// TwinCAT 3 PLC project BMS_PTM
// ProgramVersion: 3.1.4023.0
// libraries:
//   EfficientIO Communicator, * (EfficientIO)
//   Lynus Energy Basic, * (Lynus AG)
//   Lynus Energy ModbusTCP, * (Lynus AG)
//   Lynus Persistent Data V1, * (Lynus AG)
//   Lynus Standards, * (Lynus AG)
//   Tc2_ModbusSrv, * (Beckhoff Automation GmbH)
//   Tc2_Standard, * (Beckhoff Automation GmbH)
//   Tc2_System, * (Beckhoff Automation GmbH)
//   Tc2_Utilities, * (Beckhoff Automation GmbH)
//   Tc3_IotBase, * (Beckhoff Automation GmbH)
//   Tc3_Module, * (Beckhoff Automation GmbH)
// project tree:
//   / FastTask.TcTTO (not stored), MiddleTask.TcTTO, SlowTask.TcTTO (not stored)
//   FB/ FB_BatteryInverter_T.TcPOU, FB_Convert_Huawei_SmartLogger.TcPOU (not stored) (excluded from build), FB_EMS_T.TcPOU, FB_EMS_T_1.TcPOU (excluded from build), FB_EM_Beckhoff_KL3403.TcPOU (not stored), FB_Huawei_SmartLogger_1.TcPOU (excluded from build), FB_IntervalBit.TcPOU (not stored), FB_MqttCommunicator_V2_1.TcPOU (not stored), FB_Xelectrix_Powerbox_T.TcPOU
//   POUs/ prgAD.TcPOU, prgBattery.TcPOU, prgComEffIO.TcPOU, prgGrid.TcPOU, prgEMS.TcPOU, prgHouse.TcPOU, prgPersistent.TcPOU, prgPV.TcPOU, prgRWEffIO.TcPOU, prgVarEffIO.TcPOU (not stored), prg_SystemTime.TcPOU (not stored)
// real-time tasks:
//   TASK FastTask: cycle T#5ms, priority 19, ADS port 350
//   TASK MiddleTask: cycle T#10ms, priority 20, ADS port 351
//   TASK SlowTask: cycle T#20ms, priority 21, ADS port 352
// I/O:
//   DEVICE Device 1 (Beckhoff CCAT)
//   DEVICE Device 2 (CX-BK)
//     Box 1 (CX-BK)
// variable links:
//   BMS_PTM/BMS_PTM Instance <-> Device 2 (CX-BK)/Box 1 (CX-BK)
//     MiddleTask Inputs/prgGrid.fbEM1.fbKL3403.byStateCH1 <-> Term 2 (KL3403)/Channel 1/State
//     MiddleTask Inputs/prgGrid.fbEM1.fbKL3403.byStateCH2 <-> Term 2 (KL3403)/Channel 2/State
//     MiddleTask Inputs/prgGrid.fbEM1.fbKL3403.byStateCH3 <-> Term 2 (KL3403)/Channel 3/State
//     MiddleTask Inputs/prgGrid.fbEM1.fbKL3403.iDataInCH1 <-> Term 2 (KL3403)/Channel 1/Data In
//     MiddleTask Inputs/prgGrid.fbEM1.fbKL3403.iDataInCH2 <-> Term 2 (KL3403)/Channel 2/Data In
//     MiddleTask Inputs/prgGrid.fbEM1.fbKL3403.iDataInCH3 <-> Term 2 (KL3403)/Channel 3/Data In
//     MiddleTask Inputs/prgGrid.fbKBusState.uiKBusState_OUT <-> Inputs/State
//     MiddleTask Outputs/prgGrid.fbEM1.fbKL3403.byCntrCH1 <-> Term 2 (KL3403)/Channel 1/Ctrl
//     MiddleTask Outputs/prgGrid.fbEM1.fbKL3403.byCntrCH2 <-> Term 2 (KL3403)/Channel 2/Ctrl
//     MiddleTask Outputs/prgGrid.fbEM1.fbKL3403.byCntrCH3 <-> Term 2 (KL3403)/Channel 3/Ctrl

CONFIGURATION BMS_PTM
    RESOURCE PLC ON TwinCAT3
        TASK MiddleTask(INTERVAL := T#10ms, PRIORITY := 20);
        PROGRAM prgBattery WITH MiddleTask : prgBattery;
        PROGRAM prgGrid WITH MiddleTask : prgGrid;
        PROGRAM prgHouse WITH MiddleTask : prgHouse;
        PROGRAM prgPersistent WITH MiddleTask : prgPersistent;
        PROGRAM prgEMS WITH MiddleTask : prgEMS;
        PROGRAM prgPV WITH MiddleTask : prgPV;
        PROGRAM prgAD WITH MiddleTask : prgAD;
    END_RESOURCE
END_CONFIGURATION

// ---- POUs/prgBattery.TcPOU
PROGRAM prgBattery
VAR PERSISTENT
	bEnableBattery				: BOOL;							//{#lynus.ag#()}
	byPrioBattery				: BYTE;							//{#lynus.ag#()}
	lrMaxCapacityBattery		: LREAL;						//{#lynus.ag#()}
	lrCounterBattProd			: LREAL;						//{#lynus.ag#()}
	lrCounterBattCons			: LREAL;						//{#lynus.ag#()}
END_VAR
VAR
	fbBattery					: FB_Xelectrix_Powerbox_T;
	fbBattCounter				: FB_EnergyCounter;
	bIsEnabledBattery			: BOOL;							//{#lynus.ag#()}
	bResetBattery				: BOOL;							//{#lynus.ag#()}
	bSResetBattery				: BOOL;							//{#lynus.ag#()}
	byErrorWarningBattery		: BYTE;							//{#lynus.ag#()}
	dwSOCBattery				: DWORD;						//{#lynus.ag#()}
	rTargetPowerBattery			: REAL;							//{#lynus.ag#()}
	lrPowerBattery				: LREAL;						//{#lynus.ag#()}
	lrActualCapacityBattery		: LREAL;						//{#lynus.ag#()}
	lrEnergyConsumption			: LREAL;						//{#lynus.ag#()}
	lrEnergyProduction			: LREAL;						//{#lynus.ag#()}
	mTest: BOOL;

	lrPowerBattery2				: LREAL;
	lrPowerBattery3				: LREAL;						

	int_GridState: INT;											//{#lynus.ag#()}
	int_BatteryState: INT;										//{#lynus.ag#()}
	int_OperatingState: INT;									//{#lynus.ag#()}
	int_ErrorState: INT;										//{#lynus.ag#()}

	FB_Interval: FB_IntervalBit;
	m_IslandOperationStart: BOOL;								//{#lynus.ag#()}
	m_IslandOperationOngoing: BOOL;								//{#lynus.ag#()}
	m_IslandOperationStop: BOOL;								//{#lynus.ag#()}
	t_Interval :TIME:=T#30M;
	t_HightTime :TIME:=T#1S;
	
	
	m_BatteryErrorActive: BOOL;									//{#lynus.ag#()}
	m_BatteryModbusCommError: BOOL;								//{#lynus.ag#()}
	m_BatteryTargetSPError: BOOL;								//{#lynus.ag#()}
	Ton_Delay_BatteryError: Ton;
	Ton_Delay_BatteryModbusError: Ton;
	Ton_Delay_BatterySPError: Ton;
END_VAR

IF mtest THEN
	Lynus_Standards.GVL_Energy.stDataOfBatteryInverters[1,1].rTargetPowerEMS:=0;
	mtest:=FALSE;
 END_IF
 
fbBattery(
	bEnable:= bEnableBattery, 
	bActivateControl:= TRUE, 
	byUnitID:= 1, 
	byPriority:= byPrioBattery, 
	diNrOfEMS_IN:= prgEMS.fbEMS.diNrOfEMS_OUT, 
	lrMaxCapacityBattery:= lrMaxCapacityBattery, 
	sIPAdress:= '192.168.66.240', 						// modify IP Adress
	bReset:= bResetBattery, 
	stDataXelectrix=> , 
	stDataBatt=> , 
	stDataBattInverter=> , 
	stDataEMPower_Grid=> , 
	stDataEMCounter_Grid=> , 
	diNrOfBatt_OUT=> , 
	diNrOfBattInverter_OUT=> , 
	diNrOfEM_OUT_Grid=> , 
	lrMaxCapacityBattery_OUT=> );
	
//Out
bIsEnabledBattery 		:= fbBattery.stDataBatt.bEnabled;
bSResetBattery			:= fbBattery.stDataBattInverter.bStateReset;
dwSOCBattery 			:= fbBattery.stDataBatt.dwSOC;
rTargetPowerBattery 	:= fbBattery.stDataBattInverter.rTargetPower;
lrPowerBattery 			:= fbBattery.stDataBatt.lrPower;
lrActualCapacityBattery := fbBattery.lrMaxCapacityBattery_OUT;	
byErrorWarningBattery 	:= fbBattery.stDataBatt.byErrorWarning;
lrEnergyConsumption		:= fbBattery.fbEMGrid.lrTotalCounterEnergy_Consumption;
lrEnergyProduction		:= fbBattery.fbEMGrid.lrTotalCounterEnergy_Production;					
lrPowerBattery2			:= fbBattery.fbEMGrid.lrPowerTotal/1000;
							
// EnergyCounter
fbBattCounter(
	byActiveTariff:= 1, 
	lrPowerInput:= lrPowerBattery, 
	lrTotalCounterEnergy_Consumption=> , 
	lrTotalCounterEnergy_Production=> , 
	lrCounterEnergyT1_Consumption=> , 
	lrCounterEnergyT2_Consumption=> , 
	lrCounterEnergyT1_Production=> , 
	lrCounterEnergyT2_Production=> );
	
IF fbBattCounter.lrTotalCounterEnergy_Production > lrCounterBattProd THEN  	
	lrCounterBattProd := fbBattCounter.lrTotalCounterEnergy_Production;
END_IF

IF fbBattCounter.lrTotalCounterEnergy_Consumption > lrCounterBattCons THEN  	
	lrCounterBattCons := fbBattCounter.lrTotalCounterEnergy_Consumption;
END_IF

// send e states to cloud
int_GridState 		:= fbBattery.stDataXelectrix.eGridState;
int_BatteryState	:= fbBattery.stDataXelectrix.eBatteryState;
int_OperatingState	:= fbBattery.stDataXelectrix.eOperatingState;
int_ErrorState		:= fbBattery.stDataXelectrix.eErrorState;


// create bits when battery is in island operation

FB_Interval(
	m_Input			:=  prgBattery.fbBattery.stDataXelectrix.eGridState = 2,	//   2 = Island Mode 
	t_Interval 		:= t_Interval , 
	t_HighTime		:= t_HightTime, 
	m_RisingEdge	=> m_IslandOperationStart, 
	m_Interval		=> m_IslandOperationOngoing, 
	m_FallingEdge	=> m_IslandOperationStop);

// monitoring Battery status

Ton_Delay_BatteryError (In := fbBattery.stDataXelectrix.eErrorState =2,
						PT :=T#5S,
						Q => m_BatteryErrorActive);

Ton_Delay_BatteryModbusError (	In := fbBattery.stDataXelectrix.eErrorState = 1,
								PT :=T#10M,
								Q => m_BatteryModbusCommError);						

Ton_Delay_BatterySPError (	In := ABS(fbBattery.iSetpointPower/10-lrPowerBattery) > 20 AND fbBattery.stDataXelectrix.eGridState<>2 AND fbBattery.stDataBatt.dwSOC<90,	// not alarming during island operation
							PT :=T#1M,
							Q => m_BatteryTargetSPError);

END_PROGRAM

// ---- FB/FB_Xelectrix_Powerbox_T.TcPOU
FUNCTION_BLOCK FB_Xelectrix_Powerbox_T
VAR_INPUT PERSISTENT
	bEnable							: BOOL;											//{#lynus.ag#()} //True = Function is enabled, FALSE = Function is dissabled, no new Data
	bActivateControl				: BOOL;											//Activate the control from the Xelectrix Inverter over Modbus TCP (False = Inverter work by himself)
	byUnitID						: BYTE;											//Unit ID fromt the Inverter (0 to 255)
	byPriority						: BYTE;											//{#lynus.ag#()} //Priority of the Device
	diNrOfEMS_IN					: DINT;											//Number of EMS what control this Device.
	lrMaxCapacityBattery			: LREAL;										//{#lynus.ag#()} //Max Capacity from the Battery in kWh. Here on this Function this Input Value cames from Inside of the Function.
	sIPAdress						: STRING(15);									//IP Adress from the Inverter
END_VAR
VAR_INPUT
	bReset							: BOOL;											//{#lynus.ag#()} //Reset the device after a Error or a Warning
END_VAR
VAR_OUTPUT
	stDataXelectrix					: ST_Xelectrix_Powerbox_OutData;				//Shows the specific output data from the Xelectric device
	stDataBatt						: ST_Battery_Output;							//{#lynus.ag#()} //Output structure with Data from Battery
	stDataBattInverter				: ST_BatteryInverter_Output;					//{#lynus.ag#()} //Output structure with Data from Battery Inverter
	stDataEMPower_Grid				: ST_ElectricMeter_Output_Power;				//Output structure with Data from Electric Meter Grid (Power Data)
	stDataEMCounter_Grid			: ST_ElectricMeter_Output_Counter;				//Output structure with Data from Electric Meter Grid (Counter Data)
	diNrOfBatt_OUT					: DINT;											//Active Number from the Battery Function for using on other functions
	diNrOfBattInverter_OUT			: DINT;											//Active Number from the Battery Inverter Function for using on other functions
	diNrOfEM_OUT_Grid				: DINT;											//Active Number from the Electric Meter for using on other functions
	lrMaxCapacityBattery_OUT		: LREAL;										//Max kWh from the Battery system. The Xelectrix System deliver this value.
END_VAR
VAR

	fbBattery						: FB_Battery;									//Function block for battery

	fbBatteryInverter				: FB_BatteryInverter_T;							//Function block for battery inveter

	fbEMGrid						: FB_ElectricMeter;								//Electric Meter Function 

	fbPIDChrgStandby				: FB_PID;										//Controller to control the battery current on 0 in the standby mode	

	fbNumberDeviceBattery			: FB_NumberOfDevice;							//Function block to calcualte the number of the Device

	fbNumberDeviceBatteryInvert		: FB_NumberOfDevice;							//Function block to calcualte the number of the Device

	fbNumberDeviceGrid				: FB_NumberOfDevice;							//Function block to calcualte the number of the Device

	fbMBRead_FC3					: FB_MBReadRegs;								//Modbus Read Function (FC3)

	fbMBWrite_FC16					: FB_MBWriteRegs;								//Modbus Write Function (FC16)

	fbConvertData					: FB_CV_WORD_TO_DWORD;							//Convert 2 Words in a Dword

	timDelay						: TON;											//Timer for Delay between Requests

	timTimeout						: TON;											//Timer for Timeout

	timDissableFunctions			: TON;											//Timer to dissable the Function after Lynus_Standards.Constants_General.tTimeDissableLynusFunctions Days without connection to the Lynus Cloud

	timResetConnectionOnGVL			: TON;											//Timer to try reset the connection Flag on the GVL. (When somebody delete the Connection Function and make only a onlinechange)

	timReset						: TON;											//Timer to reset the Inverter after a Error

	timErrorMTCP					: TON;											//Delay when Error on Modbus TCP

	timSetStandbyCntrl				: TOF;											//Timer to set the Standby Controller

	FPEnable						: R_TRIG;										//Internal positive Edge

	FPError_FC_3					: R_TRIG;										//Internal positive Edge

	FPError_FC_16					: R_TRIG;										//Internal positive Edge

	FPActivateControl				: R_TRIG;										//Internal positive Edge

	FNTimDissable					: F_TRIG;										//Internal negative Edge

	PD_String						: FB_PersistentData_String;						//Function to save persistent data

	arrPD							: ARRAY[1..7] OF FB_PersistentData_Number;		//Function to save persistent data

	arrBuffer_FC3					: ARRAY[1..48] OF WORD;							//Buffer with Data from FC3

	arrBuffer_FC16					: ARRAY[1..2] OF WORD;							//Buffer with Data from FC16

	arrCounterForGVL				: ARRAY[1..3] OF DINT;							//Counter to clean old data on GVL

	bEnergyGridConsReceived			: BOOL;											//Energy Consumption from Grid first time received

	bEnergyGridProdReceived			: BOOL;											//Energy Production from Grid first time received

	byWaitInStep					: BYTE;											//Wait in Step before start to clean data on PLC

	byLPWorkAroundACDevice			: BYTE;											//Loop for Workaround

	byNumberOfZero					: BYTE;											//Number with 0 Value from AC Messurement

	iSetpointPower					: INT;											//Power Setpoint in W

	iStateGVLData					: INT;											//State machine to handle the data on the GVL

	iStateModbusRead				: INT;											//State variable for Statemachine

	iStateModbusWrite				: INT;											//State variable for Statemachine

	iStateModbusError				: INT;											//State variable for Statemachine

	iStateModbus_CP					: INT;											//Compare State variable

	iMaxDcDischargeCurrentBattery	: INT;											//Variable to convert from negative to positive value

	diLPForGVL						: DINT;											//Loop to clean old data on GVL

	lrEnergyGridConsumption_CP		: LREAL;										//Energy Consumption from Grid for calculation for Workaround why Xelectrix send sometimes big value 

	lrEnergyGridProduction_CP		: LREAL;										//Energy Production from Grid for calculation for Workaround why Xelectrix send sometimes big value 
	realTemp: REAL;
END_VAR
VAR PERSISTENT
	{attribute 'conditionalshow'}
	diNrOfEMS_IN_CP					: DINT;											//Number of EMS what control this Device to compare with the original
END_VAR

//Creator : Kai Ebensperger
//Company : Lynus AG
//Date : 30.06.2021
//Version : 1.0.0.0

//With this function its possible to read out values from the Xelectrix Powerbox from the factory Xelectrix
//Its also possible to controll the power in and out from Battery if its necessary.
//The protocol to the Inverter/powerbox is Modbus TCP
//When this Function is not enabled, then the Inverter is not off. But no power flows into or out of the battery.
//This Inverter deliver also the Grid power (smart Meter).
//Versions that are supported : 106
//NOTE : This Function block not support the complete emergency power mode. He switch not off when the byMaxDepthOfDischargeEPO is reached because this make the inverter by himself.

//NOTE for diNr.....Designation => 
//_IN = Here Data come in from other Functions or go out to other functions about the GVL
//_OUT = Here Data go out to other functions about the GVL

(*------------------------------------------------------------------------------------------General Input Part---------------------------------------------------------------------------------------------*)

//Check limitation
diNrOfEMS_IN := LIMIT(0,diNrOfEMS_IN,Constants_Energy.diMaxNumberOfEMS);
	
(*-------------------------------------------------------------Calcualte the number of Battery system---------------------------------------------------------------*)

fbNumberDeviceBattery(
	diActualNumberOfDevices:= Lynus_Standards.GVL_Energy.stNumberOfDevices.diNumberOfBatterys, 
	diMaxNumberOfDevices:= Constants_Energy.diMaxNumberOfBatterys, 
	udiCounterOnlineChange:= TwinCAT_SystemInfoVarList._AppInfo.OnlineChangeCnt, 
	bNumberIsCalculatet=> , 
	bFPNumberIsCalculatet=> , 
	bOnlineChange=> , 
	diNumberForThisDevice=> diNrOfBatt_OUT, 
	diNumberOfTotalDevices=> );

//Write new Numer on GVL
IF fbNumberDeviceBattery.bFPNumberIsCalculatet THEN
	Lynus_Standards.GVL_Energy.stNumberOfDevices.diNumberOfBatterys := fbNumberDeviceBattery.diNumberOfTotalDevices;	
END_IF

//Delete old Number on GVL
IF fbNumberDeviceBattery.bOnlineChange THEN 
	Lynus_Standards.GVL_Energy.stNumberOfDevices.diNumberOfBatterys := diNrOfBatt_OUT;	
		iStateGVLData := 1; 
END_IF

fbNumberDeviceBatteryInvert(
	diActualNumberOfDevices:= Lynus_Standards.GVL_Energy.stNumberOfDevices.diNumberOfBatteryInverters, 
	diMaxNumberOfDevices:= Constants_Energy.diMaxNumberOfBatteryInverters, 
	udiCounterOnlineChange:= TwinCAT_SystemInfoVarList._AppInfo.OnlineChangeCnt, 
	bNumberIsCalculatet=> , 
	bFPNumberIsCalculatet=> , 
	bOnlineChange=> , 
	diNumberForThisDevice=> diNrOfBattInverter_OUT, 
	diNumberOfTotalDevices=> );

//Write new Numer on GVL
IF fbNumberDeviceBatteryInvert.bFPNumberIsCalculatet THEN
	Lynus_Standards.GVL_Energy.stNumberOfDevices.diNumberOfBatteryInverters := fbNumberDeviceBatteryInvert.diNumberOfTotalDevices;	
END_IF

//Delete old Number on GVL
IF fbNumberDeviceBatteryInvert.bOnlineChange THEN 
	Lynus_Standards.GVL_Energy.stNumberOfDevices.diNumberOfBatteryInverters := diNrOfBattInverter_OUT;	
		iStateGVLData := 1; 
END_IF

fbNumberDeviceGrid(
	diActualNumberOfDevices:= Lynus_Standards.GVL_Energy.stNumberOfDevices.diNumberOfElectricMeters, 
	diMaxNumberOfDevices:= Constants_Energy.diMaxNumberOfElectricMeters, 
	udiCounterOnlineChange:= TwinCAT_SystemInfoVarList._AppInfo.OnlineChangeCnt, 
	bNumberIsCalculatet=> , 
	bFPNumberIsCalculatet=> , 
	bOnlineChange=> , 
	diNumberForThisDevice=> diNrOfEM_OUT_Grid, 
	diNumberOfTotalDevices=> );

//Write new Numer on GVL
IF fbNumberDeviceGrid.bFPNumberIsCalculatet THEN
	Lynus_Standards.GVL_Energy.stNumberOfDevices.diNumberOfElectricMeters := fbNumberDeviceGrid.diNumberOfTotalDevices;	
END_IF			

(*-------------------------------------------------------------Service from Backend is ready and check the connection to backend for dissabel/enable Function---------------------------------------------------------------*)

//Try to reset the variable for connection on the GVL. When all is normal then the Lynus Mqtt connection function set this variable to true in the next cycle
//When we have no connection to the backend then after Lynus_Standards.Constants_General.tTimeDissableLynusFunctions days the Function is dissabled with all of his functionalities
timResetConnectionOnGVL(IN:= NOT timResetConnectionOnGVL.Q, PT:= T#1H, Q=> , ET=> );
	IF timResetConnectionOnGVL.Q THEN Lynus_Standards.GVL_Communicator.bStateConnectionToEnableFunctions := FALSE; END_IF
		IF NOT Lynus_Standards.GVL_Communicator.bStateConnectionToEnableFunctions THEN timDissableFunctions.IN := TRUE; ELSE timDissableFunctions.IN := FALSE; END_IF  
			timDissableFunctions(IN:= , PT:= Lynus_Standards.Constants_General.tTimeDissableLynusFunctions, Q=> , ET=> );
			
(*------------------------------------------------------------------------------------------State Machine Read---------------------------------------------------------------------------------------------*)

//When the function is not enabled then the fronius control by himself without modbus tcp connection
IF NOT bEnable OR timDissableFunctions.Q THEN bActivateControl := FALSE; END_IF

//Start the Statemachine
FPEnable(CLK:= bEnable, Q=> );
	FPActivateControl(CLK:= bActivateControl, Q=> );
		FNTimDissable(CLK:= timDissableFunctions.Q, Q=> );
			IF (FPEnable.Q AND iStateModbusRead = 0 AND iStateModbusRead = 0 AND iStateModbusError = 0) OR
				(bEnable AND FPActivateControl.Q AND iStateModbusRead = 0 AND iStateModbusRead = 0 AND iStateModbusError = 0) OR
					(bEnable AND FNTimDissable.Q AND iStateModbusRead = 0 AND iStateModbusRead = 0 AND iStateModbusError = 0) THEN 
						iStateModbusRead := 1; 
			END_IF
				IF NOT bEnable OR NOT bActivateControl THEN iStateModbusRead := 0; iStateModbusWrite := 0; iStateModbusError := 0; END_IF

//Timer for delay
timDelay(IN:= , PT:= T#500MS, Q=> , ET=> );

//Timer for Timeout in Statemachine
IF (iStateModbusRead > 0 AND iStateModbusRead <= 2 AND iStateModbusRead = iStateModbus_CP) OR
		(iStateModbusWrite > 0 AND iStateModbusWrite <= 1 AND iStateModbusWrite = iStateModbus_CP) THEN
			timTimeout.IN := TRUE;
ELSE	
			timTimeout.IN := FALSE;
END_IF 
	IF iStateModbusRead = 0 AND iStateModbusWrite = 0 THEN timTimeout.IN := FALSE; END_IF
		timTimeout(IN:= , PT:= T#20S, Q=> , ET=> );

CASE iStateModbusRead OF
	
	0://Init State
		iStateModbus_CP := 0;
			timDelay.IN := FALSE;
			
		stDataXelectrix.eBatteryState := E_Xelectrix_BatteryState.eNoDataReceived;
			stDataXelectrix.eGridState := E_Xelectrix_GridState.eNoDataReceived;
				stDataXelectrix.eOperatingState := E_Xelectrix_OperatingState.eNoDataReceived;	
					stDataXelectrix.bFunctionIsActive := FALSE;
			
		fbMBRead_FC3.bExecute := FALSE;
			fbMBWrite_FC16.bExecute := FALSE;	

	1://Read all the Data
		stDataXelectrix.bFunctionIsActive := TRUE;
			iStateModbus_CP := iStateModbusRead;
		
		//Reset Write
		fbMBWrite_FC16.bExecute := FALSE;
			arrBuffer_FC16[1] := 0; arrBuffer_FC16[2] := 0;
		
		//Start Read
		fbMBRead_FC3.nQuantity := 48;
			fbMBRead_FC3.nMBAddr := 0;
				fbMBRead_FC3.bExecute := TRUE;
			
		IF fbMBRead_FC3.bBusy THEN timDelay.IN := TRUE; END_IF
		
		//Wait for Delay, copy Data and then next step
		IF NOT fbMBRead_FC3.bBusy AND NOT fbMBRead_FC3.bError AND timDelay.Q THEN
			//Grid State
			IF arrBuffer_FC3[1] = 0 THEN stDataXelectrix.eGridState := E_Xelectrix_GridState.eOff; 
			ELSIF arrBuffer_FC3[1] = 1 THEN stDataXelectrix.eGridState := E_Xelectrix_GridState.eIslandMode;
			ELSIF arrBuffer_FC3[1] = 2 THEN stDataXelectrix.eGridState := E_Xelectrix_GridState.eOnline;
			ELSIF arrBuffer_FC3[1] = 3 THEN stDataXelectrix.eGridState := E_Xelectrix_GridState.eError;   	
			END_IF
			
			(*------------------------------------------Workaround why AC device deliver sometimes 0 Value--------------------------------------------------------*)
			byNumberOfZero := 0;
				FOR byLPWorkAroundACDevice := 6 TO 9 BY 1 DO
					IF arrBuffer_FC3[byLPWorkAroundACDevice] = 0 THEN byNumberOfZero := byNumberOfZero + 1; END_IF  
				END_FOR

			IF byNumberOfZero = 0 THEN
				//Real Power (Scale factor is * 100 for W)
				fbEMGrid.lrPowerTotal := INT_TO_LREAL(WORD_TO_INT(arrBuffer_FC3[2])) * 100;
				//Reactive Power (Scale factor is * 100 for var)
				fbEMGrid.lrReactivePowerTotal := INT_TO_LREAL(WORD_TO_INT(arrBuffer_FC3[3])) * 100; 
				//Frequency (Scale factor is / 100 for Hz)
				fbEMGrid.lrFrequency := INT_TO_LREAL(WORD_TO_INT(arrBuffer_FC3[6])) / 100;
				//Voltage L1/N (Scale factor is / 10 for V)
				fbEMGrid.lrVoltageL1N := INT_TO_LREAL(WORD_TO_INT(arrBuffer_FC3[7])) / 10;
				//Voltage L2/N (Scale factor is / 10 for V)
				fbEMGrid.lrVoltageL2N := INT_TO_LREAL(WORD_TO_INT(arrBuffer_FC3[8])) / 10;
				//Voltage L3/N (Scale factor is / 10 for V)
				fbEMGrid.lrVoltageL3N := INT_TO_LREAL(WORD_TO_INT(arrBuffer_FC3[9])) / 10;
				//Current L1 (Scale factor is * 100 for mA)
				fbEMGrid.lrCurrentL1 := INT_TO_LREAL(WORD_TO_INT(arrBuffer_FC3[10])) * 100;
					//Make / 1000 for A
					fbEMGrid.lrCurrentL1 := fbEMGrid.lrCurrentL1 / 1000;
				//Current L2 (Scale factor is * 100 for mA)
				fbEMGrid.lrCurrentL2 := INT_TO_LREAL(WORD_TO_INT(arrBuffer_FC3[11])) * 100;
					//Make / 1000 for A
					fbEMGrid.lrCurrentL2 := fbEMGrid.lrCurrentL2 / 1000;
				//Current L3 (Scale factor is * 100 for mA)
				fbEMGrid.lrCurrentL3 := INT_TO_LREAL(WORD_TO_INT(arrBuffer_FC3[12])) * 100;
					//Make / 1000 for A
					fbEMGrid.lrCurrentL3 := fbEMGrid.lrCurrentL3 / 1000;
			END_IF	
			(*-----------------------------------------------------------------------------------------------------------------------------------------------------*)
			
			//Max Charge Power (Scale factor is * 100 for W)
			fbBatteryInverter.rMaxChargePowerBattInverter := INT_TO_REAL(WORD_TO_INT(arrBuffer_FC3[14])) * 100; 
			//Max Discharge Power (Scale factor is * 100 for W)
			fbBatteryInverter.rMaxDischargePowerBattInverter := INT_TO_REAL(WORD_TO_INT(arrBuffer_FC3[15])) * 100;  
				
				//SOC (No Scalefactor. Is %)	
				fbBattery.dwBatterySOC := INT_TO_DWORD(WORD_TO_INT(arrBuffer_FC3[21]));
					fbBatteryInverter.dwBatterSOC := INT_TO_DWORD(WORD_TO_INT(arrBuffer_FC3[21]));
				//Battery Temperature (Scale factor is / 100 for °C)
				fbBattery.lrBatteryTemp := INT_TO_LREAL(WORD_TO_INT(arrBuffer_FC3[23])) / 100; 
				//Battery State
				IF arrBuffer_FC3[24] = 0 THEN stDataXelectrix.eBatteryState := E_Xelectrix_BatteryState.eOff;
				ELSIF arrBuffer_FC3[24] = 1 THEN stDataXelectrix.eBatteryState := E_Xelectrix_BatteryState.eStartUp;
				ELSIF arrBuffer_FC3[24] = 2 THEN stDataXelectrix.eBatteryState := E_Xelectrix_BatteryState.eBalancing;
				ELSIF arrBuffer_FC3[24] = 3 THEN stDataXelectrix.eBatteryState := E_Xelectrix_BatteryState.eReady;
				ELSIF arrBuffer_FC3[24] = 4 THEN stDataXelectrix.eBatteryState := E_Xelectrix_BatteryState.eOperating;
				ELSIF arrBuffer_FC3[24] = 6 THEN stDataXelectrix.eBatteryState := E_Xelectrix_BatteryState.eError;
				END_IF  
				//Operating State
				IF arrBuffer_FC3[25] = 0 THEN stDataXelectrix.eOperatingState := E_Xelectrix_OperatingState.eOff;
				ELSIF arrBuffer_FC3[25] = 1 THEN stDataXelectrix.eOperatingState := E_Xelectrix_OperatingState.eDischarge;
				ELSIF arrBuffer_FC3[25] = 2 THEN stDataXelectrix.eOperatingState := E_Xelectrix_OperatingState.eCharge;
				ELSIF arrBuffer_FC3[25] = 3 THEN stDataXelectrix.eOperatingState := E_Xelectrix_OperatingState.eIdle;
				END_IF
				//Battery Capacity in Wh (Scale factor is * 100 for Wh), but make the calculation for kWh
				lrMaxCapacityBattery_OUT := arrBuffer_FC3[26] * 100;
					lrMaxCapacityBattery_OUT := lrMaxCapacityBattery_OUT / 1000;
				//Battery Current (Scale factor is * 100 for mA)
				fbBattery.lrBatteryCurrent := INT_TO_LREAL(WORD_TO_INT(arrBuffer_FC3[27])) * 100;
					//Make / 1000 for A
					fbBattery.lrBatteryCurrent := fbBattery.lrBatteryCurrent / 1000;
						//Change the sign because in view from the Battery - is discharge and + is charge. But we use vice versa	
						fbBattery.lrBatteryCurrent := fbBattery.lrBatteryCurrent * - 1; 
				//Battery Voltage 
				fbBattery.rBatteryVoltage := INT_TO_REAL(WORD_TO_INT(arrBuffer_FC3[28]));
				//Max Charge Current (Scale factor is * 100 for mA)
				fbBattery.rMaxDcChargeCurrentBattery := INT_TO_REAL(WORD_TO_INT(arrBuffer_FC3[29])) * 100; 
					//Make / 1000 for A
					fbBattery.rMaxDcChargeCurrentBattery := fbBattery.rMaxDcChargeCurrentBattery / 1000;
				//Max Discharge Current (Scale factor is * 100 for mA)
				//Its allways a negative raw value
				iMaxDcDischargeCurrentBattery := WORD_TO_INT(arrBuffer_FC3[30]);
					iMaxDcDischargeCurrentBattery := iMaxDcDischargeCurrentBattery * - 1;
						fbBattery.rMaxDcDischargeCurrentBattery := INT_TO_REAL(iMaxDcDischargeCurrentBattery) * 100; 
						realTemp := INT_TO_REAL(iMaxDcDischargeCurrentBattery) * 100; 
					//Make / 1000 for A
					fbBattery.rMaxDcDischargeCurrentBattery := fbBattery.rMaxDcDischargeCurrentBattery / 1000;
					
			(*------------------------------------------Workaround why AC device deliver sometimes 0 Value--------------------------------------------------------*)
						//Total Production (Scale factor is * 100 for Wh)
						IF byNumberOfZero = 0 THEN 
							fbConvertData(wInputValue_1:= arrBuffer_FC3[41], wInputValue_2:= arrBuffer_FC3[42], eByteOrderForConvert:= eByteOrder.eBigEndian, dwOutputValue=> );
								//Check the difference why Xelectrix send sometimes to big value
								lrEnergyGridConsumption_CP :=  DWORD_TO_LREAL((fbConvertData.dwOutputValue * 100)) / 1000 - stDataEMCounter_Grid.lrTotalCounterEnergy_Consumption; 
									IF (lrEnergyGridConsumption_CP < 15 AND fbConvertData.dwOutputValue <> 0) OR NOT bEnergyGridConsReceived THEN 
										fbEMGrid.lrCounterEnergyT1_Consumption := fbConvertData.dwOutputValue * 100;
											fbEMGrid.lrCounterEnergyT1_Consumption := fbEMGrid.lrCounterEnergyT1_Consumption / 1000;
												fbEMGrid.lrTotalCounterEnergy_Consumption := fbEMGrid.lrCounterEnergyT1_Consumption;
									END_IF
										IF DWORD_TO_LREAL((fbConvertData.dwOutputValue * 100)) / 1000 <> 0 AND NOT bEnergyGridConsReceived THEN bEnergyGridConsReceived := TRUE; END_IF 
							//Total Consumption (Scale factor is * 100 for Wh)
							fbConvertData(wInputValue_1:= arrBuffer_FC3[43], wInputValue_2:= arrBuffer_FC3[44], eByteOrderForConvert:= eByteOrder.eBigEndian, dwOutputValue=> );
								//Check the difference why Xelectrix send sometimes to big value
								 lrEnergyGridProduction_CP :=  DWORD_TO_LREAL((fbConvertData.dwOutputValue * 100)) / 1000 - stDataEMCounter_Grid.lrTotalCounterEnergy_Production;
									IF (lrEnergyGridProduction_CP < 15 AND fbConvertData.dwOutputValue <> 0) OR NOT bEnergyGridProdReceived THEN 
										fbEMGrid.lrCounterEnergyT1_Production := fbConvertData.dwOutputValue * 100;
											fbEMGrid.lrCounterEnergyT1_Production := fbEMGrid.lrCounterEnergyT1_Production / 1000;
												fbEMGrid.lrTotalCounterEnergy_Production := fbEMGrid.lrCounterEnergyT1_Production;
									END_IF
										IF DWORD_TO_LREAL((fbConvertData.dwOutputValue * 100)) / 1000 <> 0 AND NOT bEnergyGridProdReceived THEN bEnergyGridProdReceived := TRUE; END_IF 
						END_IF
			(*-----------------------------------------------------------------------------------------------------------------------------------------------------*)		
						
			//Go to Next Step
			fbMBRead_FC3.bExecute := FALSE;
				timDelay.IN := FALSE;		
					iStateModbusRead := 2;
		END_IF
		
		//Xelectrics Grid Error
		IF NOT fbMBRead_FC3.bBusy AND NOT fbMBRead_FC3.bError AND timDelay.Q AND stDataXelectrix.eGridState = E_Xelectrix_GridState.eError THEN
			iStateModbusError := 300;
				stDataXelectrix.eErrorState := E_Xelectrix_Error.eXelectrixError;
		END_IF
			//Xelectrics Battery Error
			IF NOT fbMBRead_FC3.bBusy AND NOT fbMBRead_FC3.bError AND timDelay.Q AND stDataXelectrix.eBatteryState = E_Xelectrix_BatteryState.eError THEN
				iStateModbusError := 300;
					stDataXelectrix.eErrorState := E_Xelectrix_Error.eXelectrixError;
			END_IF
		
		//Error or Timeout
		IF FPError_FC_3.Q OR timTimeout.Q THEN
			iStateModbusError := 300;
				stDataXelectrix.eErrorState := E_Xelectrix_Error.eModbusTCPError;
		END_IF
	
	2://Wait 1 Step to reset the delay counter befor start to write
		iStateModbus_CP := iStateModbusRead;
		
			iStateModbusWrite := 1;
				iStateModbusRead := - 1;	
				
		//Timeout
		IF timTimeout.Q THEN
			iStateModbusError := 300;
				stDataXelectrix.eErrorState := E_Xelectrix_Error.eModbusTCPError;
		END_IF
		
END_CASE

(*----------------------------------------------------------------------------------------Battery Inverter Function----------------------------------------------------------------------------------------------*)

//Error and Reset
timErrorMTCP(IN:= stDataXelectrix.bError AND stDataXelectrix.eErrorState = E_Xelectrix_Error.eModbusTCPError, PT:= T#5S, Q=> , ET=> );

IF timDissableFunctions.Q THEN fbBatteryInverter.bWarning := TRUE; fbBatteryInverter.iWarningCode := 0; ELSE fbBatteryInverter.bWarning := FALSE; END_IF 
	IF (stDataXelectrix.bError AND stDataXelectrix.eBatteryState = E_Xelectrix_BatteryState.eError) OR timErrorMTCP.Q OR Lynus_Standards.GVL_Energy.stNumberOfDevices.diNumberOfBatteryInverters > Constants_Energy.diMaxNumberOfBatteryInverters THEN fbBatteryInverter.bError := TRUE; ELSE fbBatteryInverter.bError := FALSE; END_IF	
		IF Lynus_Standards.GVL_Energy.stNumberOfDevices.diNumberOfBatteryInverters > Constants_Energy.diMaxNumberOfBatteryInverters THEN fbBatteryInverter.iErrorCode := 1;
		ELSIF stDataXelectrix.bError THEN fbBatteryInverter.iErrorCode := 0; 
		END_IF  

//Autoreset after Error, because Xelectrix deleiver somtimes a Error and they dont know why.....
timReset(IN:= stDataBattInverter.byErrorWarning <> 0 AND NOT timReset.Q, PT:= T#1S, Q=> , ET=> );	
		
//Island mode active
IF stDataXelectrix.eGridState = E_Xelectrix_GridState.eIslandMode THEN fbBatteryInverter.bWorkOnIslandMode := TRUE; ELSE fbBatteryInverter.bWorkOnIslandMode := FALSE; END_IF
		
//Function
fbBatteryInverter(
	bEnable:= bEnable AND NOT timDissableFunctions.Q, 
	bInverterOnOff:= TRUE, 
	bError:= , 
	bWarning:= , 
	bReset:= bReset OR timReset.Q,  
	bWorkOnIslandMode:= , 
	bWriteWithDelay:= TRUE, 
	byPriority:= byPriority, 
	byReserveSOCEPO:= Lynus_Standards.GVL_Energy.stDataOfBatteryInverters[diNrOfEMS_IN,diNrOfBattInverter_OUT].byReserveSOCEPO, 
	byMaxDepthOfDischargeEPO:= Lynus_Standards.GVL_Energy.stDataOfBatteryInverters[diNrOfEMS_IN,diNrOfBattInverter_OUT].byMaxDepthOfDischargeEPO, 
	iErrorCode:= , 
	iWarningCode:= , 
	dwBatterSOC:= , 
	rTargetPower:= Lynus_Standards.GVL_Energy.stDataOfBatteryInverters[diNrOfEMS_IN,diNrOfBattInverter_OUT].rTargetPowerEMS, 
	lrActualBatteryPower:= fbBattery.lrBatteryCurrent * fbBattery.rBatteryVoltage, 
	rMaxChargePowerBattInverter:= , 
	rMaxDischargePowerBattInverter:= , 
	lrBattInverterPowerOnIslandMode:= 0, 
	lrBattInverterPowerOnNormalMode:= 0, 
	tTimDelayOutput:= T#5S, 
	stDataBattInvertOut=> , 
	stDataBattInvertOutDelay=> stDataBattInverter);

//Controller to hold the Battery Current to 0 and take the rest from the Grid. (Avoid discharge in standby or when reaching the reserve charge for EPO)
timSetStandbyCntrl(IN:= fbBatteryInverter.stDataBattInvertOut.rTargetPower = 0, PT:= T#5S, Q=> , ET=> );

IF timSetStandbyCntrl.Q AND bEnable AND bActivateControl THEN
	fbPIDChrgStandby.bEnable := TRUE;
		//Charge the Battery when its under the reserve for SOC
		IF fbBatteryInverter.dwBatterSOC < fbBatteryInverter.byReserveSOCEPO THEN
			fbPIDChrgStandby.rSetpoint := (fbBattery.stDataBatteryOut.rMaxDcChargeCurrent * 0.1) * - 1; 	
		ELSE
			fbPIDChrgStandby.rSetpoint := 0;	
		END_IF		 
ELSE
	fbPIDChrgStandby.bEnable := FALSE;
END_IF

fbPIDChrgStandby( 
	bEnable:= , 
	rSetpoint:= , 
	udiIValue:= 750, 
	udiDValue:= 0, 
	udiDamping:= 0, 
	rPValue:= 0.32, 
	rMaxValue:= 0, 
	rMinValue:= ((fbBatteryInverter.rMaxChargePowerBattInverter / 100) * - 1) / 2, 
	rNeutralZone:= 0.1, 
	bDirection:= FALSE, 
	rActualValue:= LREAL_TO_REAL(fbBattery.stDataBatteryOut.lrCurrent), 
	rQController=> );	

//Set the Target power to a fixed value when the controller is acitve
IF fbPIDChrgStandby.bEnable THEN 
	stDataBattInverter.rTargetPower := - 1;
END_IF
	
(*----------------------------------------------------------------------------------------Battery Function----------------------------------------------------------------------------------------------*)

//Error
IF timDissableFunctions.Q THEN fbBattery.bWarning := TRUE; fbBattery.iWarningCode := 0; ELSE fbBattery.bWarning := FALSE; END_IF 
	IF (stDataXelectrix.bError AND stDataXelectrix.eBatteryState = E_Xelectrix_BatteryState.eError) OR timErrorMTCP.Q OR Lynus_Standards.GVL_Energy.stNumberOfDevices.diNumberOfBatterys > Constants_Energy.diMaxNumberOfBatterys THEN fbBattery.bError := TRUE; ELSE fbBattery.bError := FALSE; END_IF
		IF Lynus_Standards.GVL_Energy.stNumberOfDevices.diNumberOfBatterys > Constants_Energy.diMaxNumberOfBatterys THEN fbBattery.iErrorCode := 1;
		ELSIF stDataXelectrix.bError THEN fbBattery.iErrorCode := 0; 
		END_IF

//Function
fbBattery(
	bEnable:= bEnable AND NOT timDissableFunctions.Q, 
	bError:= , 
	bWarning:= , 
	bCalculatePower:= TRUE, 
	bReset:= bReset OR timReset.Q, 
	bWriteWithDelay:= TRUE, 
	iErrorCode:= , 
	iWarningCode:= , 
	dwBatterySOC:= , 
	dwBatterySOH:= 0, 
	rBatteryVoltage:= , 
	rMaxDcChargeCurrentBattery:= , 
	rMaxDcDischargeCurrentBattery:= , 
	rMaxChargeVoltage:= 0, 
	lrMaxCapacityBattery:= lrMaxCapacityBattery, 
	lrBatteryPower:= 0, 
	lrBatteryCurrent:= , 
	lrBatteryTemp:= , 
	tTimDelayOutput:= T#5S, 
	stDataBatteryOut=> , 
	stDataBatteryOutDelay=> stDataBatt);

(*----------------------------------------------------------------------------------------Electric Meter Function for Grid----------------------------------------------------------------------------------------------*)

//Error
IF timDissableFunctions.Q THEN fbEMGrid.bWarning := TRUE; fbEMGrid.iWarningCode := 0; ELSE fbEMGrid.bWarning := FALSE; END_IF 
	IF (stDataXelectrix.bError AND stDataXelectrix.eGridState = E_Xelectrix_GridState.eError) OR timErrorMTCP.Q OR Lynus_Standards.GVL_Energy.stNumberOfDevices.diNumberOfElectricMeters > Constants_Energy.diMaxNumberOfElectricMeters THEN fbEMGrid.bError := TRUE; ELSE fbEMGrid.bError := FALSE; END_IF
		IF Lynus_Standards.GVL_Energy.stNumberOfDevices.diNumberOfElectricMeters > Constants_Energy.diMaxNumberOfElectricMeters THEN fbEMGrid.iErrorCode := 1;
		ELSIF stDataXelectrix.bError THEN fbEMGrid.iErrorCode := 0;
		END_IF  

//Read Out Data done for EM Function
IF iStateModbusRead <> 1 THEN fbEMGrid.bReadOutDataDone := TRUE; ELSE fbEMGrid.bReadOutDataDone := FALSE; END_IF		
		
//Function
fbEMGrid(
	bEnable:= bEnable AND NOT timDissableFunctions.Q, 
	bError:= , 
	bEnableReadOutFunction:= FALSE, 
	bWriteWithDelay:= TRUE, 
	bPowerDataInvers:= FALSE,
	bReadOutDataDone:= ,
	iTimeReadOutInterval:= , 
	iErrorCode:= , 
	iWarningCode:= , 
	lrTotalCounterEnergy_Consumption:= , 
	lrTotalCounterEnergy_Production:= , 
	lrCounterEnergyT1_Consumption:= , 
	lrCounterEnergyT2_Consumption:= 0, 
	lrCounterEnergyT1_Production:= , 
	lrCounterEnergyT2_Production:= 0, 
	lrCurrentL1:= , 
	lrVoltageL1N:= , 
	lrVoltageL1L2:= 0, 
	lrPowerL1:= 0, 
	lrCurrentL2:= , 
	lrVoltageL2N:= , 
	lrVoltageL2L3:= 0, 
	lrPowerL2:= 0, 
	lrCurrentL3:= , 
	lrVoltageL3N:= , 
	lrVoltageL3L1:= 0, 
	lrPowerL3:= 0, 
	lrPowerTotal:= , 
	lrFrequency:= , 
	lrReactivePowerTotal:= , 
	lrApparentPowerTotal:= 0, 
	tTimDelayOutput:= T#5S, 
	stDataEMOutPower=> , 
	stDataEMOutPowerDelay=> stDataEMPower_Grid, 
	stDataEMOutCounter=> ,
	stDataEMOutCounterDelay=> stDataEMCounter_Grid,  
	bReadOutMeter=> );

(*------------------------------------------------------------------------------------------State Machine Write---------------------------------------------------------------------------------------------*)	
	
CASE iStateModbusWrite OF	
	
	1://Setpoint for Power and set the Timout on Inverter to 10 Seconds. (When after this time the inverter not received a new Message over Modbus TCP, then he goes back in his own automatic mode and work by himself)
		iStateModbus_CP := iStateModbusWrite;	
		
		fbMBWrite_FC16.nQuantity := 2;
			fbMBWrite_FC16.nMBAddr := 100;
				fbMBWrite_FC16.bExecute := TRUE;
		
		//Setpoint for the Power when discharge (Scale factor is / 100 for W on the Inverter) 
		IF fbBatteryInverter.stDataBattInvertOut.rTargetPower >= 0 THEN
			IF ((fbBatteryInverter.stDataBattInvertOut.rMaxDischargePower * 1000) * (fbBatteryInverter.stDataBattInvertOut.rTargetPower / 100)) / 100 >= - 32768 AND 
				((fbBatteryInverter.stDataBattInvertOut.rMaxDischargePower * 1000) * (fbBatteryInverter.stDataBattInvertOut.rTargetPower / 100)) / 100 <= 32767 THEN
					iSetpointPower := REAL_TO_INT(((fbBatteryInverter.stDataBattInvertOut.rMaxDischargePower * 1000) * (fbBatteryInverter.stDataBattInvertOut.rTargetPower / 100)) / 100);  
						arrBuffer_FC16[1] := INT_TO_WORD(iSetpointPower);
			END_IF
		END_IF
		//Setpoint for the Power when charge (Scale factor is / 100 for W on the Inverter) 
		IF fbBatteryInverter.stDataBattInvertOut.rTargetPower < 0 OR fbPIDChrgStandby.bEnable THEN
			IF ((fbBatteryInverter.stDataBattInvertOut.rMaxChargePower * 1000) * (fbBatteryInverter.stDataBattInvertOut.rTargetPower / 100)) / 100 >= - 32768 AND 
				((fbBatteryInverter.stDataBattInvertOut.rMaxChargePower * 1000) * (fbBatteryInverter.stDataBattInvertOut.rTargetPower / 100)) / 100 <= 32767 THEN
					iSetpointPower := REAL_TO_INT(((fbBatteryInverter.stDataBattInvertOut.rMaxChargePower * 1000) * (fbBatteryInverter.stDataBattInvertOut.rTargetPower / 100)) / 100);  
						//Take the Setpoint from the Standby Controller
						IF fbPIDChrgStandby.bEnable AND fbPIDChrgStandby.rQController <= 0 AND fbPIDChrgStandby.rQController >= -32768 THEN
							iSetpointPower := REAL_TO_INT(fbPIDChrgStandby.rQController);  
						END_IF
					arrBuffer_FC16[1] := INT_TO_WORD(iSetpointPower); 
			END_IF
		END_IF
		//Timeout Time
		arrBuffer_FC16[2] := 10;
		
		IF fbMBWrite_FC16.bBusy THEN timDelay.IN := TRUE; END_IF

		//Wait for Delay and then next step
		IF NOT fbMBWrite_FC16.bBusy AND NOT fbMBWrite_FC16.bError AND timDelay.Q THEN
			fbMBWrite_FC16.bExecute := FALSE;
				timDelay.IN := FALSE;
					stDataXelectrix.bError := FALSE; 
						stDataXelectrix.eErrorState := E_Xelectrix_Error.eNoError;
							//Restart from new with the Read out part
							iStateModbusRead := 1;
								iStateModbusWrite := 0;
		END_IF
				
		//Error or Timout
		IF FPError_FC_16.Q OR timTimeout.Q THEN
			iStateModbusError := 300;
				stDataXelectrix.eErrorState := E_Xelectrix_Error.eModbusTCPError;
		END_IF

END_CASE

(*------------------------------------------------------------------------------------------State Machine Write---------------------------------------------------------------------------------------------*)	

CASE iStateModbusError OF
	
	300://Error
		iStateModbus_CP := iStateModbusError;
			timDelay.IN := FALSE;
				fbMBRead_FC3.bExecute := FALSE;
					fbMBWrite_FC16.bExecute := FALSE;
						stDataXelectrix.bError := TRUE;	
							//Restart from new with the Read out part after an Error
							iStateModbusRead := 1;	
								iStateModbusError := 0;
									iStateModbusWrite := 0;
END_CASE

(*------------------------------------------------------------------------------------------Modbus TCP Functions---------------------------------------------------------------------------------------------*)

fbMBRead_FC3(sIPAddr:= sIPAdress, nUnitID := byUnitID, nTCPPort:= 502, cbLength:= SIZEOF(arrBuffer_FC3), pDestAddr:= ADR(arrBuffer_FC3), tTimeout:= T#10S );
	FPError_FC_3(CLK:= fbMBRead_FC3.bError, Q=> );

fbMBWrite_FC16(sIPAddr:= sIPAdress, nTCPPort:= 502, nUnitID := byUnitID, cbLength:= SIZEOF(arrBuffer_FC16), pSrcAddr:= ADR(arrBuffer_FC16), tTimeout:= T#10S );
	FPError_FC_16(CLK:= fbMBWrite_FC16.bError, Q=> );

(*-----------------------------------------------------------Handle data to Global structure for al Devices that are included in this function-----------------------------------------------------------------*)

//Delete al old Data on GVL after a online change or change on the variable diNrOfEMS_IDOD
IF diNrOfEMS_IN <> diNrOfEMS_IN_CP AND iStateGVLData = 0 THEN iStateGVLData := 10; END_IF 

CASE iStateGVLData OF
	
	0://Init Step
		byWaitInStep := 0;
			arrCounterForGVL[1] := 1; arrCounterForGVL[2] := 1; arrCounterForGVL[3] := 1;
	
	1://Wait for 4 Steps before clean al Data on GVL
		byWaitInStep := byWaitInStep + 1;
			IF (byWaitInStep >= 4 AND (fbNumberDeviceBattery.bNumberIsCalculatet OR fbNumberDeviceBatteryInvert.bNumberIsCalculatet OR fbNumberDeviceGrid.bNumberIsCalculatet)) THEN iStateGVLData := 2; END_IF
				//To much Devices, back to the Init step
				IF byWaitInStep >= 4 AND NOT fbNumberDeviceBattery.bNumberIsCalculatet AND NOT fbNumberDeviceBatteryInvert.bNumberIsCalculatet AND NOT fbNumberDeviceGrid.bNumberIsCalculatet THEN iStateGVLData := 0; END_IF	
			
	2://Clear all Data in GVL
		FOR diLPForGVL := 1 TO Constants_Energy.diMaxNumberOfEMS BY 1 DO
			//Battery Inverters 
			IF fbNumberDeviceBatteryInvert.bNumberIsCalculatet THEN 
				Lynus_Standards.GVL_Energy.stDataOfBatteryInverters[diLPForGVL,arrCounterForGVL[1]].bEnabled := FALSE;
					Lynus_Standards.GVL_Energy.stDataOfBatteryInverters[diLPForGVL,arrCounterForGVL[1]].bOnOff := FALSE;
						Lynus_Standards.GVL_Energy.stDataOfBatteryInverters[diLPForGVL,arrCounterForGVL[1]].bWorkOnIslandMode := FALSE;
							Lynus_Standards.GVL_Energy.stDataOfBatteryInverters[diLPForGVL,arrCounterForGVL[1]].byErrorWarning := 0;
								Lynus_Standards.GVL_Energy.stDataOfBatteryInverters[diLPForGVL,arrCounterForGVL[1]].byPriority := 0;
									Lynus_Standards.GVL_Energy.stDataOfBatteryInverters[diLPForGVL,arrCounterForGVL[1]].dwBatterySOC := 0;
										Lynus_Standards.GVL_Energy.stDataOfBatteryInverters[diLPForGVL,arrCounterForGVL[1]].lrPowerOnIslandMode := 0;
											Lynus_Standards.GVL_Energy.stDataOfBatteryInverters[diLPForGVL,arrCounterForGVL[1]].rMaxChargePower := 0;
												Lynus_Standards.GVL_Energy.stDataOfBatteryInverters[diLPForGVL,arrCounterForGVL[1]].rMaxDischargePower := 0;
													Lynus_Standards.GVL_Energy.stDataOfBatteryInverters[diLPForGVL,arrCounterForGVL[1]].lrPowerNormalMode := 0;
														//Set also the target value from ems back here to 0 and not in EMS function because EMS is in Standy when we have a online change (Problem when we delete a ems function and make a online change)
														Lynus_Standards.GVL_Energy.stDataOfBatteryInverters[diLPForGVL,arrCounterForGVL[1]].rTargetPowerEMS := 0;
															Lynus_Standards.GVL_Energy.stDataOfBatteryInverters[diLPForGVL,arrCounterForGVL[1]].byMaxDepthOfDischargeEPO := 0;
																Lynus_Standards.GVL_Energy.stDataOfBatteryInverters[diLPForGVL,arrCounterForGVL[1]].byReserveSOCEPO := 0;
			END_IF
				//Batterys 
				IF fbNumberDeviceBattery.bNumberIsCalculatet THEN 
					Lynus_Standards.GVL_Energy.stDataOfBatterys[diLPForGVL,arrCounterForGVL[2]].bEnabled := FALSE;
						Lynus_Standards.GVL_Energy.stDataOfBatterys[diLPForGVL,arrCounterForGVL[2]].byErrorWarning := 0;
							Lynus_Standards.GVL_Energy.stDataOfBatterys[diLPForGVL,arrCounterForGVL[2]].dwSOC := 0;
								Lynus_Standards.GVL_Energy.stDataOfBatterys[diLPForGVL,arrCounterForGVL[2]].dwSOH := 0;
									Lynus_Standards.GVL_Energy.stDataOfBatterys[diLPForGVL,arrCounterForGVL[2]].lrCapacity := 0;
										Lynus_Standards.GVL_Energy.stDataOfBatterys[diLPForGVL,arrCounterForGVL[2]].lrCurrent := 0;
											Lynus_Standards.GVL_Energy.stDataOfBatterys[diLPForGVL,arrCounterForGVL[2]].lrPower := 0;
												Lynus_Standards.GVL_Energy.stDataOfBatterys[diLPForGVL,arrCounterForGVL[2]].lrPowerConsumption := 0;
													Lynus_Standards.GVL_Energy.stDataOfBatterys[diLPForGVL,arrCounterForGVL[2]].lrPowerProduction := 0;
														Lynus_Standards.GVL_Energy.stDataOfBatterys[diLPForGVL,arrCounterForGVL[2]].lrTemp := 0;
															Lynus_Standards.GVL_Energy.stDataOfBatterys[diLPForGVL,arrCounterForGVL[2]].rMaxChargeVoltage := 0;
																Lynus_Standards.GVL_Energy.stDataOfBatterys[diLPForGVL,arrCounterForGVL[2]].rMaxDcChargeCurrent := 0;
																	Lynus_Standards.GVL_Energy.stDataOfBatterys[diLPForGVL,arrCounterForGVL[2]].rMaxDcDischargeCurrent := 0;
																		Lynus_Standards.GVL_Energy.stDataOfBatterys[diLPForGVL,arrCounterForGVL[2]].rVoltage := 0;
				END_IF
		END_FOR
			//Electric Meter Grid
			IF fbNumberDeviceGrid.bNumberIsCalculatet THEN 
				Lynus_Standards.GVL_Energy.stDataElectricMeters[arrCounterForGVL[3]].bEnabled := FALSE;	
					Lynus_Standards.GVL_Energy.stDataElectricMeters[arrCounterForGVL[3]].byErrorWarning := 0;
						Lynus_Standards.GVL_Energy.stDataElectricMeters[arrCounterForGVL[3]].lrCounterEnergyT1_Consumption := 0;
							Lynus_Standards.GVL_Energy.stDataElectricMeters[arrCounterForGVL[3]].lrCounterEnergyT1_Production := 0;
								Lynus_Standards.GVL_Energy.stDataElectricMeters[arrCounterForGVL[3]].lrCounterEnergyT2_Consumption := 0;
									Lynus_Standards.GVL_Energy.stDataElectricMeters[arrCounterForGVL[3]].lrCounterEnergyT2_Production := 0;
										Lynus_Standards.GVL_Energy.stDataElectricMeters[arrCounterForGVL[3]].lrPower := 0;
											Lynus_Standards.GVL_Energy.stDataElectricMeters[arrCounterForGVL[3]].lrPowerConsumption := 0;
												Lynus_Standards.GVL_Energy.stDataElectricMeters[arrCounterForGVL[3]].lrPowerProduction := 0;
													Lynus_Standards.GVL_Energy.stDataElectricMeters[arrCounterForGVL[3]].lrTotalCounterEnergy_Consumption := 0;
														Lynus_Standards.GVL_Energy.stDataElectricMeters[arrCounterForGVL[3]].lrTotalCounterEnergy_Production := 0;
			END_IF
		
			//Counter for Battery Inverter
			arrCounterForGVL[1] := arrCounterForGVL[1] + 1;
				arrCounterForGVL[1] := LIMIT(0,arrCounterForGVL[1],Constants_Energy.diMaxNumberOfBatteryInverters);
			//Counter for Batterys
			arrCounterForGVL[2] := arrCounterForGVL[2] + 1;
				arrCounterForGVL[2] := LIMIT(0,arrCounterForGVL[2],Constants_Energy.diMaxNumberOfBatterys);
			//Electric Meters
			arrCounterForGVL[3] := arrCounterForGVL[3] + 1;
				arrCounterForGVL[3] := LIMIT(0,arrCounterForGVL[3],Constants_Energy.diMaxNumberOfElectricMeters);
					//Back to the init step
					IF arrCounterForGVL[1] >= Constants_Energy.diMaxNumberOfBatteryInverters AND arrCounterForGVL[2] >= Constants_Energy.diMaxNumberOfBatterys AND  
						arrCounterForGVL[3] >= Constants_Energy.diMaxNumberOfElectricMeters THEN 
							iStateGVLData := 0; 
					END_IF

	10://Clear old Data on GVL 		
		//Battery Inverter
		Lynus_Standards.GVL_Energy.stDataOfBatteryInverters[diNrOfEMS_IN_CP,diNrOfBattInverter_OUT].bEnabled := FALSE;
			Lynus_Standards.GVL_Energy.stDataOfBatteryInverters[diNrOfEMS_IN_CP,diNrOfBattInverter_OUT].bOnOff := FALSE;
				Lynus_Standards.GVL_Energy.stDataOfBatteryInverters[diNrOfEMS_IN_CP,diNrOfBattInverter_OUT].bWorkOnIslandMode := FALSE;
					Lynus_Standards.GVL_Energy.stDataOfBatteryInverters[diNrOfEMS_IN_CP,diNrOfBattInverter_OUT].byErrorWarning := 0;
						Lynus_Standards.GVL_Energy.stDataOfBatteryInverters[diNrOfEMS_IN_CP,diNrOfBattInverter_OUT].byPriority := 0;
							Lynus_Standards.GVL_Energy.stDataOfBatteryInverters[diNrOfEMS_IN_CP,diNrOfBattInverter_OUT].dwBatterySOC := 0;
								Lynus_Standards.GVL_Energy.stDataOfBatteryInverters[diNrOfEMS_IN_CP,diNrOfBattInverter_OUT].lrPowerOnIslandMode := 0;
									Lynus_Standards.GVL_Energy.stDataOfBatteryInverters[diNrOfEMS_IN_CP,diNrOfBattInverter_OUT].rMaxChargePower := 0;
										Lynus_Standards.GVL_Energy.stDataOfBatteryInverters[diNrOfEMS_IN_CP,diNrOfBattInverter_OUT].rMaxDischargePower := 0;
											Lynus_Standards.GVL_Energy.stDataOfBatteryInverters[diNrOfEMS_IN_CP,diNrOfBattInverter_OUT].lrPowerNormalMode := 0;
		//Batterys		
		Lynus_Standards.GVL_Energy.stDataOfBatterys[diNrOfEMS_IN_CP,diNrOfBatt_OUT].bEnabled := FALSE;
			Lynus_Standards.GVL_Energy.stDataOfBatterys[diNrOfEMS_IN_CP,diNrOfBatt_OUT].byErrorWarning := 0;
				Lynus_Standards.GVL_Energy.stDataOfBatterys[diNrOfEMS_IN_CP,diNrOfBatt_OUT].dwSOC := 0;
					Lynus_Standards.GVL_Energy.stDataOfBatterys[diNrOfEMS_IN_CP,diNrOfBatt_OUT].dwSOH := 0;
						Lynus_Standards.GVL_Energy.stDataOfBatterys[diNrOfEMS_IN_CP,diNrOfBatt_OUT].lrCapacity := 0;
							Lynus_Standards.GVL_Energy.stDataOfBatterys[diNrOfEMS_IN_CP,diNrOfBatt_OUT].lrCurrent := 0;
								Lynus_Standards.GVL_Energy.stDataOfBatterys[diNrOfEMS_IN_CP,diNrOfBatt_OUT].lrPower := 0;
									Lynus_Standards.GVL_Energy.stDataOfBatterys[diNrOfEMS_IN_CP,diNrOfBatt_OUT].lrPowerConsumption := 0;
										Lynus_Standards.GVL_Energy.stDataOfBatterys[diNrOfEMS_IN_CP,diNrOfBatt_OUT].lrPowerProduction := 0;
											Lynus_Standards.GVL_Energy.stDataOfBatterys[diNrOfEMS_IN_CP,diNrOfBatt_OUT].lrTemp := 0;
												Lynus_Standards.GVL_Energy.stDataOfBatterys[diNrOfEMS_IN_CP,diNrOfBatt_OUT].rMaxChargeVoltage := 0;
													Lynus_Standards.GVL_Energy.stDataOfBatterys[diNrOfEMS_IN_CP,diNrOfBatt_OUT].rMaxDcChargeCurrent := 0;
														Lynus_Standards.GVL_Energy.stDataOfBatterys[diNrOfEMS_IN_CP,diNrOfBatt_OUT].rMaxDcDischargeCurrent := 0;
															Lynus_Standards.GVL_Energy.stDataOfBatterys[diNrOfEMS_IN_CP,diNrOfBatt_OUT].rVoltage := 0;
									
		diNrOfEMS_IN_CP := diNrOfEMS_IN;
			//Back to the init step
			iStateGVLData := 0;

END_CASE 	 

//Write Data on GVL for Battery Inverter
IF diNrOfBattInverter_OUT > 0 AND fbNumberDeviceBatteryInvert.bNumberIsCalculatet AND diNrOfEMS_IN > 0 THEN
	Lynus_Standards.GVL_Energy.stDataOfBatteryInverters[diNrOfEMS_IN,diNrOfBattInverter_OUT].bEnabled := fbBatteryInverter.stDataBattInvertOut.bEnabled;
		Lynus_Standards.GVL_Energy.stDataOfBatteryInverters[diNrOfEMS_IN,diNrOfBattInverter_OUT].bOnOff := fbBatteryInverter.stDataBattInvertOut.bOnOff;
			Lynus_Standards.GVL_Energy.stDataOfBatteryInverters[diNrOfEMS_IN,diNrOfBattInverter_OUT].bWorkOnIslandMode := fbBatteryInverter.stDataBattInvertOut.bWorkOnIslandMode;
				Lynus_Standards.GVL_Energy.stDataOfBatteryInverters[diNrOfEMS_IN,diNrOfBattInverter_OUT].byErrorWarning := fbBatteryInverter.stDataBattInvertOut.byErrorWarning;
					Lynus_Standards.GVL_Energy.stDataOfBatteryInverters[diNrOfEMS_IN,diNrOfBattInverter_OUT].byPriority := fbBatteryInverter.stDataBattInvertOut.byPriority;
						Lynus_Standards.GVL_Energy.stDataOfBatteryInverters[diNrOfEMS_IN,diNrOfBattInverter_OUT].dwBatterySOC := fbBatteryInverter.dwBatterSOC;
							Lynus_Standards.GVL_Energy.stDataOfBatteryInverters[diNrOfEMS_IN,diNrOfBattInverter_OUT].lrPowerOnIslandMode := fbBatteryInverter.stDataBattInvertOut.lrPowerOnIslandMode;	
								Lynus_Standards.GVL_Energy.stDataOfBatteryInverters[diNrOfEMS_IN,diNrOfBattInverter_OUT].rMaxChargePower := fbBatteryInverter.stDataBattInvertOut.rMaxChargePower;
									Lynus_Standards.GVL_Energy.stDataOfBatteryInverters[diNrOfEMS_IN,diNrOfBattInverter_OUT].rMaxDischargePower := fbBatteryInverter.stDataBattInvertOut.rMaxDischargePower;
										Lynus_Standards.GVL_Energy.stDataOfBatteryInverters[diNrOfEMS_IN,diNrOfBattInverter_OUT].lrPowerNormalMode := fbBatteryInverter.stDataBattInvertOut.lrPowerNormalMode;	
END_IF 
	//Write Data on GVL for Batterys
	IF diNrOfBatt_OUT > 0 AND fbNumberDeviceBattery.bNumberIsCalculatet AND diNrOfEMS_IN > 0 THEN
		Lynus_Standards.GVL_Energy.stDataOfBatterys[diNrOfEMS_IN,diNrOfBatt_OUT].bEnabled := fbBattery.stDataBatteryOut.bEnabled;	
			Lynus_Standards.GVL_Energy.stDataOfBatterys[diNrOfEMS_IN,diNrOfBatt_OUT].byErrorWarning := fbBattery.stDataBatteryOut.byErrorWarning;
				Lynus_Standards.GVL_Energy.stDataOfBatterys[diNrOfEMS_IN,diNrOfBatt_OUT].dwSOC := fbBattery.stDataBatteryOut.dwSOC;
					Lynus_Standards.GVL_Energy.stDataOfBatterys[diNrOfEMS_IN,diNrOfBatt_OUT].dwSOH := fbBattery.stDataBatteryOut.dwSOH;
						Lynus_Standards.GVL_Energy.stDataOfBatterys[diNrOfEMS_IN,diNrOfBatt_OUT].lrCapacity := fbBattery.stDataBatteryOut.lrCapacity;
							Lynus_Standards.GVL_Energy.stDataOfBatterys[diNrOfEMS_IN,diNrOfBatt_OUT].lrCurrent := fbBattery.stDataBatteryOut.lrCurrent;
								Lynus_Standards.GVL_Energy.stDataOfBatterys[diNrOfEMS_IN,diNrOfBatt_OUT].lrPower := fbBattery.stDataBatteryOut.lrPower;
									Lynus_Standards.GVL_Energy.stDataOfBatterys[diNrOfEMS_IN,diNrOfBatt_OUT].lrPowerConsumption := fbBattery.stDataBatteryOut.lrPowerConsumption;
										Lynus_Standards.GVL_Energy.stDataOfBatterys[diNrOfEMS_IN,diNrOfBatt_OUT].lrPowerProduction := fbBattery.stDataBatteryOut.lrPowerProduction;
											Lynus_Standards.GVL_Energy.stDataOfBatterys[diNrOfEMS_IN,diNrOfBatt_OUT].lrTemp := fbBattery.stDataBatteryOut.lrTemp;
												Lynus_Standards.GVL_Energy.stDataOfBatterys[diNrOfEMS_IN,diNrOfBatt_OUT].rMaxChargeVoltage := fbBattery.stDataBatteryOut.rMaxChargeVoltage;
													Lynus_Standards.GVL_Energy.stDataOfBatterys[diNrOfEMS_IN,diNrOfBatt_OUT].rMaxDcChargeCurrent := fbBattery.stDataBatteryOut.rMaxDcChargeCurrent;
														Lynus_Standards.GVL_Energy.stDataOfBatterys[diNrOfEMS_IN,diNrOfBatt_OUT].rMaxDcDischargeCurrent := fbBattery.stDataBatteryOut.rMaxDcDischargeCurrent;
															Lynus_Standards.GVL_Energy.stDataOfBatterys[diNrOfEMS_IN,diNrOfBatt_OUT].rVoltage := fbBattery.stDataBatteryOut.rBatteryVoltage;
	END_IF
//Write Data on GVL for Electric Meter (Grid)
IF diNrOfEM_OUT_Grid > 0 AND fbNumberDeviceGrid.bNumberIsCalculatet THEN
	Lynus_Standards.GVL_Energy.stDataElectricMeters[diNrOfEM_OUT_Grid].bEnabled := fbEMGrid.stDataEMOutPower.bEnabled;
		Lynus_Standards.GVL_Energy.stDataElectricMeters[diNrOfEM_OUT_Grid].byErrorWarning := fbEMGrid.stDataEMOutPower.byErrorWarning;
			Lynus_Standards.GVL_Energy.stDataElectricMeters[diNrOfEM_OUT_Grid].lrCounterEnergyT1_Consumption := fbEMGrid.stDataEMOutCounter.lrCounterEnergyT1_Consumption;
				Lynus_Standards.GVL_Energy.stDataElectricMeters[diNrOfEM_OUT_Grid].lrCounterEnergyT1_Production := fbEMGrid.stDataEMOutCounter.lrCounterEnergyT1_Production;
					Lynus_Standards.GVL_Energy.stDataElectricMeters[diNrOfEM_OUT_Grid].lrCounterEnergyT2_Consumption := fbEMGrid.stDataEMOutCounter.lrCounterEnergyT2_Consumption;
						Lynus_Standards.GVL_Energy.stDataElectricMeters[diNrOfEM_OUT_Grid].lrCounterEnergyT2_Production := fbEMGrid.stDataEMOutCounter.lrCounterEnergyT2_Production;		
							Lynus_Standards.GVL_Energy.stDataElectricMeters[diNrOfEM_OUT_Grid].lrPower := fbEMGrid.stDataEMOutPower.lrPowerTotal;
								Lynus_Standards.GVL_Energy.stDataElectricMeters[diNrOfEM_OUT_Grid].lrPowerConsumption := fbEMGrid.stDataEMOutPower.lrPowerConsumption;
									Lynus_Standards.GVL_Energy.stDataElectricMeters[diNrOfEM_OUT_Grid].lrPowerProduction := fbEMGrid.stDataEMOutPower.lrPowerProduction;
										Lynus_Standards.GVL_Energy.stDataElectricMeters[diNrOfEM_OUT_Grid].lrTotalCounterEnergy_Consumption := fbEMGrid.stDataEMOutCounter.lrTotalCounterEnergy_Consumption;
											Lynus_Standards.GVL_Energy.stDataElectricMeters[diNrOfEM_OUT_Grid].lrTotalCounterEnergy_Production := fbEMGrid.stDataEMOutCounter.lrTotalCounterEnergy_Production;
END_IF

(*----------------------------------------------------------Save persistent data----------------------------------------------------------------*)

arrPD[1](lrValue:= BOOL_TO_LREAL(bEnable), bEventBasedActive=> );
arrPD[2](lrValue:= BOOL_TO_LREAL(bActivateControl), bEventBasedActive=> );
arrPD[3](lrValue:= BYTE_TO_LREAL(byUnitID), bEventBasedActive=> );
arrPD[4](lrValue:= BYTE_TO_LREAL(byPriority), bEventBasedActive=> );
arrPD[5](lrValue:= DINT_TO_LREAL(diNrOfEMS_IN), bEventBasedActive=> );
arrPD[6](lrValue:= lrMaxCapacityBattery, bEventBasedActive=> );
arrPD[7](lrValue:= DINT_TO_LREAL(diNrOfEMS_IN_CP), bEventBasedActive=> );
PD_String(sText:= sIPAdress, bEventBasedActive=> );

END_FUNCTION_BLOCK

// ---- FB/FB_BatteryInverter_T.TcPOU
FUNCTION_BLOCK FB_BatteryInverter_T
VAR_INPUT

	bEnable								: BOOL;								//Enable/Disable Battery Inverter

	bInverterOnOff						: BOOL;								//Switch the Inverter On or Off

	bError								: BOOL;								//Battery Inverter has a Error

	bWarning							: BOOL;								//Battery Inverter has a Warning

	bReset								: BOOL;								//Reset after the inverter switch off regarding a Error. Need also to reset the warning

	bWorkOnIslandMode					: BOOL;								//True when the inverter work in island mode

	bWriteWithDelay						: BOOL;								//Write with Delay the Data to the output (Not al Output Data is writen with Delay)

	byPriority							: BYTE; 							//Priority of the device if controlled via the EMS block => 1 2 3 (If 0 then this device does not exist for the EMS block)

	byReserveSOCEPO						: BYTE;								//Reserve SOC in battery for emergency power operation

	byMaxDepthOfDischargeEPO			: BYTE; 							//If islanding is active, the maximum discharge depth of the batteries can be set here until the inverter switches off.

	iErrorCode							: INT;								//Error Code from external Battery inverter

	iWarningCode						: INT;								//Warning Code from external Battery inverter

	dwBatterSOC							: DWORD;							//The actual Battery state of Charge

	rTargetPower						: REAL;								//Target Power from the EMS Function

	lrActualBatteryPower				: LREAL;							//Actual Battery power in W

	rMaxChargePowerBattInverter			: REAL; 							//Max. charge power battery inverter with unit W

	rMaxDischargePowerBattInverter		: REAL;								//Max. discharge power battery inverter with unit W

	lrBattInverterPowerOnIslandMode		: LREAL;							//Power from the battery inverter when island mode is active with unit W

	lrBattInverterPowerOnNormalMode		: LREAL;							//Power from the battery inverter when normal mode is active with unit W

	tTimDelayOutput						: TIME := T#5S;						//Delay Time to write some Data to the Output	
END_VAR
VAR_OUTPUT

	stDataBattInvertOut					: ST_BatteryInverter_Output;		//Batter Inverter output data

	stDataBattInvertOutDelay			: ST_BatteryInverter_Output;		//Batter Inverter output data with delay
END_VAR
VAR
	FPReset								: R_TRIG;							//Internal rising edge
	FPResetTim							: R_TRIG;							//Internal rising edge
	FPEnable							: R_TRIG;							//Internal positive Edge
	FNEnable							: F_TRIG;							//Internal negative Edge
	timReset							: TOF;								//Timer for Reset
	timStandby							: TON;								//Timer to set the inverter in standby mode
	timDisableInEPO						: TON;								//Timer do disable the inverter when work on Island mode an battery soc is under min
	timDelayOutputs						: TON;								//Timer to send Data with Delay to the outputs
	bMaxDephOfDischargeReached			: BOOL;								//True when the max of discharge in emergency power mode is reached
END_VAR

//Creator : Kai Ebensperger
//Company : Lynus AG
//Date : 18.05.2021
//Version : 1.0.0.0

//With this function is possible to control the most popular things on a battery inverter
//NOTE : With this Function its only poaaible to override the commands on a battery inverter
//All limits and important things control the inverter by himself.
//In Grid mode the Battery Inverter charge the battery to 100% SOC and discharge to 0% or to the limit for emergency power mode
//On Island mode the battery inverter charge the battery to 100% SOC. Discharge its possible to the max discharge setting. If the soc from the battery is <= this value the inverter switch off after 5 minutes when no power goes inside the battery
//With Reset you can reset the warnings and errors on the inverter.
//Also when the battery inverter is enabled by the timer for max discharge limit in emergency mode you can restart the inverter with a reset.
//When the target power for the inverter = 0 then the inverter go to the standby mode an switch off.

//---------------------------------------------------------------------Check the limits of the inputs--------------------------------------------------------------------------------------
byReserveSOCEPO := LIMIT(0,byReserveSOCEPO,100);
	byMaxDepthOfDischargeEPO := LIMIT(0,byMaxDepthOfDischargeEPO,100);
		dwBatterSOC := LIMIT(0,dwBatterSOC,100);
			rTargetPower := LIMIT(-100,rTargetPower,100);
				lrActualBatteryPower := LIMIT(-1000000,lrActualBatteryPower,1000000);
					lrBattInverterPowerOnIslandMode := LIMIT(-1000000,lrBattInverterPowerOnIslandMode,1000000);
						lrBattInverterPowerOnNormalMode := LIMIT(-1000000,lrBattInverterPowerOnNormalMode,1000000);
							rMaxChargePowerBattInverter := LIMIT(-1000000,rMaxChargePowerBattInverter,1000000);
								rMaxDischargePowerBattInverter := LIMIT(-1000000,rMaxDischargePowerBattInverter,1000000);

//---------------------------------------------------------------------------Data directly to the output-------------------------------------------------------------------------------------------
stDataBattInvertOut.byPriority := byPriority;
	stDataBattInvertOut.bEnabled := bEnable;
		stDataBattInvertOut.bWorkOnIslandMode := bWorkOnIslandMode;

//--------------------------------------------------------------------------Max Deph of discharge SOC in Emergency power mode---------------------------------------------------------------
IF dwBatterSOC <= byMaxDepthOfDischargeEPO AND lrActualBatteryPower >= 0 AND stDataBattInvertOut.bWorkOnIslandMode THEN timDisableInEPO.IN := TRUE; END_IF
	IF dwBatterSOC > byMaxDepthOfDischargeEPO OR lrActualBatteryPower < 0 OR NOT stDataBattInvertOut.bWorkOnIslandMode OR NOT stDataBattInvertOut.bOnOff OR (FPResetTim.Q AND bMaxDephOfDischargeReached) THEN timDisableInEPO.IN := FALSE; bMaxDephOfDischargeReached := FALSE; END_IF	
		timDisableInEPO(IN:= , PT:= T#5M, Q=> , ET=> );  
			IF timDisableInEPO.Q THEN bMaxDephOfDischargeReached := TRUE; END_IF		
		
//-----------------------------------------------------------------------------Reset-------------------------------------------------------------------------------------------------------
FPReset(CLK:= bReset, Q=> );
	timReset(IN:= stDataBattInvertOut.byErrorWarning <> 0 AND FPReset.Q AND NOT timReset.Q, PT:= T#2S, Q=> stDataBattInvertOut.bStateReset, ET=> );
		FPResetTim(CLK:= timReset.Q, Q=> );
			IF FPResetTim.Q THEN stDataBattInvertOut.byErrorWarning := 0; END_IF	

//--------------------------------------------------------------------------Error or Warning-------------------------------------------------------------------------------------------------
IF bWarning AND stDataBattInvertOut.byErrorWarning <> 2 THEN stDataBattInvertOut.byErrorWarning := 1; END_IF 
IF bError OR (timDisableInEPO.Q AND NOT FPResetTim.Q) THEN stDataBattInvertOut.byErrorWarning := 2; END_IF 			

//Error Codes
IF stDataBattInvertOut.byErrorWarning = 2 AND iErrorCode = 0 THEN stDataBattInvertOut.eMessage := E_Message_BatteryInverter.eBatteryInverterError;
ELSIF stDataBattInvertOut.byErrorWarning = 2 AND iErrorCode = 1 THEN stDataBattInvertOut.eMessage := E_Message_BatteryInverter.eTooMuchBatteryInverter;
ELSE stDataBattInvertOut.eMessage := E_Message_BatteryInverter.eNoMessage; 
END_IF
			
//--------------------------------------------------------------------------Target power--------------------------------------------------------------------------------------------------
stDataBattInvertOut.rTargetPower := rTargetPower;
	//Target power to 0
	IF (NOT stDataBattInvertOut.bWorkOnIslandMode AND stDataBattInvertOut.rTargetPower > 0 AND dwBatterSOC <= byReserveSOCEPO) OR
		(stDataBattInvertOut.rTargetPower < 0 AND dwBatterSOC >= 100) OR
			(NOT stDataBattInvertOut.bWorkOnIslandMode AND stDataBattInvertOut.rTargetPower > 0 AND dwBatterSOC <= 0) THEN 
				stDataBattInvertOut.rTargetPower := 0; 
	END_IF  
		//Set the Inverter in Standby	
		timStandby(IN:= stDataBattInvertOut.rTargetPower = 0 AND NOT stDataBattInvertOut.bWorkOnIslandMode, PT:= T#1M, Q=> , ET=> );
	
//--------------------------------------------------------------------Enable or disable the Inverter--------------------------------------------------------------------------------------
IF bEnable AND bInverterOnOff AND stDataBattInvertOut.byErrorWarning <> 2 THEN
	stDataBattInvertOut.bOnOff := TRUE;
END_IF			
	IF timStandby.Q OR stDataBattInvertOut.byErrorWarning = 2 OR NOT bEnable OR NOT bInverterOnOff THEN
		stDataBattInvertOut.bOnOff := FALSE;
	END_IF 				
	
//-------------------------------------------------------------------Outputs--------------------------------------------------------------------------------------------------------------
IF stDataBattInvertOut.bWorkOnIslandMode THEN 
	stDataBattInvertOut.lrPowerOnIslandMode := lrBattInverterPowerOnIslandMode / 1000;
		stDataBattInvertOut.lrPowerOnIslandMode := LINT_TO_LREAL(LREAL_TO_LINT(stDataBattInvertOut.lrPowerOnIslandMode * 100)) / 100;
			stDataBattInvertOut.lrPowerNormalMode := 0;	 
ELSE
	stDataBattInvertOut.lrPowerNormalMode := lrBattInverterPowerOnNormalMode / 1000;
		stDataBattInvertOut.lrPowerNormalMode := LINT_TO_LREAL(LREAL_TO_LINT(stDataBattInvertOut.lrPowerNormalMode * 100)) / 100; 	 
			stDataBattInvertOut.lrPowerOnIslandMode := 0;
END_IF

stDataBattInvertOut.rMaxChargePower := rMaxChargePowerBattInverter / 1000;
	stDataBattInvertOut.rMaxChargePower := DINT_TO_REAL(REAL_TO_DINT(stDataBattInvertOut.rMaxChargePower * 100)) / 100; 
	
stDataBattInvertOut.rMaxDischargePower := rMaxDischargePowerBattInverter / 1000;
	stDataBattInvertOut.rMaxDischargePower := DINT_TO_REAL(REAL_TO_DINT(stDataBattInvertOut.rMaxDischargePower * 100)) / 100; 

timDelayOutputs(IN:= bWriteWithDelay AND bEnable AND NOT timDelayOutputs.Q, PT:= tTimDelayOutput, Q=> , ET=> );
	FPEnable(CLK:= bEnable, Q=> );
		FNEnable(CLK:= bEnable, Q=> );
		
//Write with Delay or without
IF (bWriteWithDelay AND (timDelayOutputs.Q OR FPEnable.Q OR FNEnable.Q)) OR NOT bWriteWithDelay THEN
	stDataBattInvertOutDelay := stDataBattInvertOut;	
END_IF

END_FUNCTION_BLOCK

// ---- POUs/prgEMS.TcPOU
PROGRAM prgEMS
VAR PERSISTENT
	byMaxDepthOfDischrgEPO		: BYTE;							//{#lynus.ag#()}
	byPrioMinChrgBattSOCInEPO	: BYTE;							//{#lynus.ag#()}
	byResChrgfromGridToBatt		: BYTE;							//{#lynus.ag#()}
	byResChrgfromGridToBatt_Controlled		: BYTE;							//{#lynus.ag#()}
	byReserveSOCEPO				: BYTE;							//{#lynus.ag#()}
	uiUpdateTime				: UINT;							//{#lynus.ag#()}
	bEnableEMS					: BOOL;							//{#lynus.ag#()}
	bAllowChrgFromGrid			: BOOL;							//{#lynus.ag#()}
	rMainFuseCSEMS				: REAL;							//{#lynus.ag#()}
	iOperationModeEMS			: INT;							//{#lynus.ag#()}
END_VAR
VAR
	fbEMS						: FB_EMS_T;
	bIsEnableEMS				: BOOL;							//{#lynus.ag#()}
	bStateAllowChrgFromGrid		: BOOL;							//{#lynus.ag#()}
	bHPActivate					: BOOL;							//{#lynus.ag#()}
	bControllingState			: BOOL;							//{#lynus.ag#()}
	iMessageEMS					: INT;							//{#lynus.ag#()}
	rHeartbeatEMS				: REAL;							//{#lynus.ag#()}
	rErrorWarningEMS			: REAL;							//{#lynus.ag#()}
	rReadyEMS					: REAL;							//{#lynus.ag#()}
	rNewBatteryPowerEMS			: REAL;							//{#lynus.ag#()}
	b_EnableBatteryChargingControl				: BOOL:=TRUE;																						//{#lynus.ag#()} //  
	b_StartReleaseBatteryCharging				: BOOL;																								//{#lynus.ag#()} //  
	b_StopReleaseBatteryCharging				: BOOL;																								//{#lynus.ag#()} //  
	b_TimeBasedReleaseChargingBattery			: BOOL;																								//{#lynus.ag#()} //  
	b_StartChargingfor3Hours					: BOOL;																								//{#lynus.ag#()} //  

	RS_ChargingFromGridAllowed: Rs;
	tof_3HourCharging: Tof;
	RS_3HourCharging: Rs;
	r_trig_3HourChraging: R_trig;
	f_trig_3HourChragingOver: f_trig;
	m_PIDBatterySC_Enabled: BOOL;
	m_PIDBatteryPLCLM_Dischrg_Enabled: BOOL;
	m_fbPIDBatteryPLCLM_Chrg_Enabled: BOOL;
	m_fbPIDBatteryEPO_Enabled: BOOL;
END_VAR

// Stefan 21.02.2024
// disabled bControllingState to make sure the backend is not regulating the battery
// changeed lacal EMS PID regulator for charging and discharging in FB_EMS_T to fullfill the PTM requirements to fixie PID parameters, made the regulator slower for more stability. 

fbEMS.stSetupEMS.bAllowChrgFromGrid := bAllowChrgFromGrid;
fbEMS.stSetupEMS.byMaxDepthOfDischrgEPO := byMaxDepthOfDischrgEPO;
fbEMS.stSetupEMS.byPrioMinChrgBattSOCInEPO := byPrioMinChrgBattSOCInEPO;
fbEMS.stSetupEMS.byReserveSOCEPO := byReserveSOCEPO;
fbEMS.stSetupEMS.rSizeMainFuseCS := rMainFuseCSEMS;
fbEMS.stSetupEMS.uiUpdateTime := uiUpdateTime;

IF iOperationModeEMS = 0 THEN fbEMS.eOperationMode := E_OperatingMode_EMS.eAllOff;
ELSIF iOperationModeEMS = 1 THEN fbEMS.eOperationMode := E_OperatingMode_EMS.eSelfConsumption;	
ELSIF iOperationModeEMS = 2 THEN fbEMS.eOperationMode := E_OperatingMode_EMS.ePeakLoadCapping;
ELSIF iOperationModeEMS = 3 THEN fbEMS.eOperationMode := E_OperatingMode_EMS.eLoadManagement;			
END_IF

fbEMS(
	bEnable						:= bEnableEMS, 
	diNrOfEM_IN_ECS				:= , 
	stSetupEMS					:= , 
	eOperationMode				:= , 
	eSpeedModeBackendController	:= E_SpeedModeBackendController_EMS.eFast, 
	eSpeedModeLocalController	:= E_SpeedModeLocalController_EMS.eFast,
	bActivateHP					:= bHPActivate, 
	bControllingState			:= TRUE, //bControllingState, 
	rHeartbeat					:= rHeartbeatEMS, 
	rErrorWarning				:= rErrorWarningEMS, 
	rEnergyOptReady				:= rReadyEMS, 
	rNewBattPower				:= rNewBatteryPowerEMS, 
	b_ZeroPowerRegulation		:=,
	b_EnableBatteryChargingControl	:= TRUE,
	b_StartReleaseBatteryCharging 	:= TRUE,
	b_StopReleaseBatteryCharging 	:= ,
	rMaxBattChargingPower			:= SEL(bAllowChrgFromGrid,100,63),	// 80 kW = 100%, 63 % = 50 kW
	rPeakDetectionforCalculation 	:= 20,	// was original 3, caused issues that load management not caluculeted. see EMS line 313
	
	eMessageEMS				=> iMessageEMS, 
	bStateEnable			=> bIsEnableEMS, 
	bStateAllowChrgFromGrid	=> bStateAllowChrgFromGrid, 
	bMissingPowerData		=> , 
	bSurplusAvailable		=> , 
	byProgress				=> , 
	uiState_OUT				=> , 
	diNrOfEMS_OUT			=> , 
	arrMinPrioReached		=> , 
	arrMaxPrioReached		=> ,
	b_TimeBasedReleaseChargingBattery => b_TimeBasedReleaseChargingBattery);
	
	// update 20230228 
	// charging control done with bAllowChrgFromGrid: Charging is allways allowed (If surplus is available) , but charging from grid is only allowed during the night time. 
// b_EnableBatteryChargingControl
// b_StartReleaseBatteryCharging
// b_StopReleaseBatteryCharging
// fbEMS.stSetupEMS.bAllowChrgFromGrid := bAllowChrgFromGrid;
RS_ChargingFromGridAllowed( SET := b_EnableBatteryChargingControl AND b_StartReleaseBatteryCharging,
							Reset1 := NOT b_EnableBatteryChargingControl OR (b_EnableBatteryChargingControl AND b_StopReleaseBatteryCharging));

r_trig_3HourChraging( 	clk:=b_StartChargingfor3Hours);
f_trig_3HourChragingOver( clk:=tof_3HourCharging.Q);

tof_3HourCharging(	IN:= r_trig_3HourChraging.Q,
					PT := T#3H);
RS_3HourCharging(	Set := r_trig_3HourChraging.Q,
					Reset1 := f_trig_3HourChragingOver.Q OR (r_trig_3HourChraging.Q AND RS_3HourCharging.Q1) OR prgBattery.dwSOCBattery > byResChrgfromGridToBatt_Controlled);
							
							
IF b_EnableBatteryChargingControl AND (RS_ChargingFromGridAllowed.Q1 OR RS_3HourCharging.Q1) THEN
	bAllowChrgFromGrid := TRUE;
	fbEMS.stSetupEMS.byResChrgfromGridToBatt := byResChrgfromGridToBatt_Controlled; // battery max soc according input field when charging the battery in the night
ELSE
	bAllowChrgFromGrid := FALSE;
	fbEMS.stSetupEMS.byResChrgfromGridToBatt := byResChrgfromGridToBatt;			// battery max SOC according to EMS setting, e.g. 100%; this should only get achieved by grid surplus
END_IF
 
// find out which regulator is active

m_PIDBatterySC_Enabled := fbEMS.fbPIDBatterySC.bEnable;;
m_PIDBatteryPLCLM_Dischrg_Enabled := fbEMS.fbPIDBatteryPLCLM_Dischrg.bEnable;
m_fbPIDBatteryPLCLM_Chrg_Enabled := fbEMS.fbPIDBatteryPLCLM_Chrg.bEnable;
m_fbPIDBatteryEPO_Enabled := fbEMS.fbPIDBatteryEPO.bEnable;

END_PROGRAM

// ---- FB/FB_EMS_T.TcPOU
FUNCTION_BLOCK FB_EMS_T
VAR_INPUT PERSISTENT
	bEnable										: BOOL;																								//{#lynus.ag#()} //Enable and dissable this function
	diNrOfEM_IN_ECS								: DINT;																								//Number of the electric meter for incoming power data. (Its for the complete consumption of all charging stations)
	stSetupEMS									: ST_Setup_EMS := (uiUpdateTime := 15);																//{#lynus.ag#()} //Setup EMS
	eOperationMode								: E_OperatingMode_EMS;																				//{#lynus.ag#()} //Operation Mode EMS
	eSpeedModeBackendController					: E_SpeedModeBackendController_EMS;																	//Speed for the Controller what discharge the Battery when the commands come from the Backend
	eSpeedModeLocalController					: E_SpeedModeLocalController_EMS;																	//Speed for the local Controller for charge and discharge the Battery
	b_ZeroPowerRegulation						: BOOL;																								//{#lynus.ag#()} // activates the Battery discharging before using the mains during LoadManagement; Line 1728/1732/1738 
	b_EnableBatteryChargingControl				: BOOL;																								//{#lynus.ag#()} //  
	b_StartReleaseBatteryCharging				: BOOL;																								//{#lynus.ag#()} //  
	b_StopReleaseBatteryCharging				: BOOL;																								//{#lynus.ag#()} //  
END_VAR
VAR_INPUT
	bActivateHP									: BOOL;																								//{#lynus.ag#()} //Activate the Heating pumps when the Backend deliver the signal. NOT OVERRIDE
	bControllingState							: BOOL;																								//{#lynus.ag#()} //The control state of the service is linked here. NOT OVERRIDE
	rHeartbeat									: REAL;																								//{#lynus.ag#()} //Heartbeat from the Service. NOT OVERRIDE
	rErrorWarning								: REAL;																								//{#lynus.ag#()} //Error or Warning from the Service. NOT OVERRIDE
	rEnergyOptReady								: REAL;																								//{#lynus.ag#()} //Energy Optimization Service Ready. NOT OVERRIDE
	rNewBattPower								: REAL;																								//{#lynus.ag#()} //New Battery Power from Backend Service. NOT OVERRIDE
	rMaxBattChargingPower						: REAL:=100;																								// Maximum Battery Charging power in percent
	rPeakDetectionforCalculation				: REAL:=3;																								// Value for Peak detection, was original 3 but caused issues with fast changing loads (e.g. industrie)
END_VAR
VAR_OUTPUT
	eMessageEMS									: Lynus_Standards.E_Message_EMS;																	//EMS Message
	bStateEnable								: BOOL;																								//{#lynus.ag#()} //Show if the ems function is enabled or not
	bStateAllowChrgFromGrid						: BOOL;																								//{#lynus.ag#()} //Show the State if the charging from grid is allowed or not
	bMissingPowerData							: BOOL;																								//Missing data on the max power setup from one ore more devices
	bSurplusAvailable							: BOOL;																								//Variable that indicates if there is surplus or not
	byProgress									: BYTE;																								//Shows the Progress from the new Calculation when we have Surplus. When we have no Surplus and we discharge the batterys this Value is on 100
	uiState_OUT									: UINT;																								//Actual State
	diNrOfEMS_OUT								: DINT;																								//Active Number from the EMS Function for using on other functions
	arrMinPrioReached							: ARRAY[1..5] OF BOOL;																				//Shows if all different devices types are set to 0% with the target power ([1] = Battery, [2] = HP, [3] = EHE, [4] = OBC, [5] = ECS)
	arrMaxPrioReached							: ARRAY[1..5] OF BOOL;																				//Shows if all different devices types are set to 100% with the target power ([1] = Battery, [2] = HP, [3] = EHE, [4] = OBC, [5] = ECS)	
	b_TimeBasedReleaseChargingBattery			: BOOL;																								//
END_VAR	
VAR
	(*-----------------------------------------------------------------------Internal Variables and Functions for connection to the Backend--------------------------------------------------------------------------------*)
	fbPIDDischrgCmdFromBackend					: FB_PID;																							//PID Contrller what controll the discharging power from the Battery when the controlling from backend is activated
	timDissableFunctions						: TON;																								//Timer to dissable the Function after Lynus_Standards.Constants_General.tTimeDissableLynusFunctions Days without connection to the Lynus Cloud
	timResetConnectionOnGVL						: TON;																								//Timer to try reset the connection Flag on the GVL. (When somebody delete the Connection Function and make only a onlinechange)
	timHB										: TON;																								//Timer to check the Heartbeat from the Backendservice
	timPIDDischrgCmdFromBackend					: TON;																								//Timer to set the output from the pid controller to 0 due to internal control deviations (Backend Mode)
	timCorrectionSetpoint						: TOF;																								//Timer to make the correction on the Setpoint for Battery power. This is neccessary to give time to the inverter and Grid to adjust on the new values
	timErrorWarning								: TON;																								//Timer to enable the Function Backend Mode after a Error or Warning
	timEnergyOptReady							: TON;																								//Timer to enable the Function Backend Mode after the Backend Service is ready
	timControlingState							: TON;																								//Timer to enable the controlling over the Backend Mode
	timResetActivateHP							: TON;																								//Timer to reset the Activate HP Command from the Backend Service
	FPEnablePID									: R_TRIG;																							//Internal positive edge
	FPMakeCorrection							: R_TRIG;																							//Internal positive edge
	bDischrgCmdFromBackendOK					: BOOL;																								//Allowed to controll the Devices from Backend
	rHeartbeat_CP								: REAL;																								//Compare the Heartbeat from the Backend
	rControllerQPIDDischrgCmdFromBackend		: REAL;																								//Controller output from pid controll over Backend Mode
	rNewBattPower_CP							: REAL;																								//New Battery power to ckeck if we have received a new Value in kW
	lrActualPowerBatterys						: LREAL;																							//Actual Power from the Batterys in kW
	lrErrorPIDCorrectionDischrgCmdFromBackend	: LREAL;																							//Limit the Error on the pid controller for discahrge the battery on the controll over Backend Mode
	lrNewBatteryPowerWithCorrection				: LREAL;																							//The New Battery power from the Backend with correction that we dont insert power in the Grid
	liLPDischrgCmdFromBackend					: LINT;																								//Loop to send the command from Backend to the Devices
	(*-----------------------------------------------------------------------------------Rest of internal Variabels and Functions---------------------------------------------------------------------------------------*)
	fbMessagesEMS								: FB_EMS_Message;																					//FB to create the Messages for this Function
	fbNumberDevice								: FB_NumberOfDevice;																				//Function block to calcualte the number of the Device
	fbTaskIndex									: GETCURTASKINDEX;																					//Function to read out the Task Index in witch the function is running
	fbPIDBatterySC								: FB_PID;																							//PID Controller to discharge the battery in the self consumption mode
	fbPIDBatteryEPO								: FB_PID;																							//PID Controller to discharge the battery in the emergency power mode
	fbPIDBatteryPLCLM_Dischrg					: FB_PID;																							//PID Controller to Dischage the battery on load management mode and peak shaving mode
	fbPIDBatteryPLCLM_Chrg						: FB_PID;																							//PID Controller to Charge the battery on load management mode and peak shaving mode
	timCalculateNewPowerValue					: TON;																								//Timer to start a new session to calculate the new power value for the devices
	timPIDSC									: TON;																								//Timer to set the output from the pid controller to 0 due to internal control deviations (Self consumption mode)
	timPIDEPO									: TON;																								//Timer to set the output from the pid controller to 0 due to internal control deviations (Emergency power mode)
	timCorrectionECS							: TON;																								//Timer for make the correction for ECS in the Load management and peak capping mode with use the separate fuse
	timErrorGridMessurement						: TON;																								//Timer with delay to stop the EMS Function if we have a error on the Grid messurement
	timTimeout									: TON;																								//Timer for Timout
	timCutPeaks									: TOF;																								//Timer to cut peaks on the grid. The system waits for this time for strong and short peaks before regulating.
	timDelayStart								: TOF;																								//Timer with the delay to start the ems function after a online change
	timResetDisableECS							: TOF;																								//Timer to reset the dissbling the ECS after a Error from the Electric Meter what messure the power from all ECS
	FPEPO										: R_TRIG;																							//Internal positive edge
	FNEPO										: F_TRIG;																							//Internal negative edge
	eOperationModeEMS_CP						: E_OperatingMode_EMS;																				//Operation Mode EMS/Battery to compare with the original variable
	arrPD										: ARRAY[1..12] OF FB_PersistentData_Number;															//Function to save persistent data
	arrTimBatterysAreFull						: ARRAY[1..Constants_Energy.diMaxNumberOfBatteryInverters] OF TON;									//Timer start for each Battery when is full
	arrActualStepInTurn_CP						: ARRAY[1..2] OF BYTE;																				//Actual Step in turn to compare with original variable
	arrActualPrioInTurn							: ARRAY[1..5] OF BYTE;																				//Actual Priority (1-255) that is currently in turn ([1] = Battery, [2] = HP, [3] = EHE, [4] = OBC, [5] = ECS)
	arrActualStepInTurn							: ARRAY[1..2] OF BYTE;																				//Actual Step (1-10) from step switched devices that is currently in turn ([1] = HP, [2] = EHE)
	arrLPPrioZeroSetToZeroP						: ARRAY[1..5] OF LINT;																				//Array with loop to set each device with priority 0 to the target power value 
	arrCTCheckActivePrio						: ARRAY[1..5] OF LINT;																				//Array with loop to check the actual prioritys
	bEPMActive									: BOOL;																								//Emergency power mode is active
	bChargePrioBatterysOnEPO					: BOOL;																								//Load batterys that made a island grid first to the adjustable SOC before start with al other devices
	bStepWasOn100								: BOOL;																								//Its true when the actual step from step switched devices was on 100%
	bECSPrio255									: BOOL;																								//True when we reached the max prio of the charging stations
	bStopAll									: BOOL;																								//Stop the EMS when we some is happend what make trouble
	bDisableECS									: BOOL;																								//Dissable the ECS when the EM what messure the power from all ECS has a error
	bErrorOnGridMessurement						: BOOL;																								//Shows if on the Grid Messurement is a error and stop then the EMS Function
	bNoPowerForECS								: BOOL;																								//Variable what shows that we dont can give more power on the ECS because we have to much power on the Fuse line on wich the ECS is connected
	bySmGrActiveCommonPrio_CP					: BYTE;																								//Smalest or greatest active common priority of the devices to compare with the original varible
	byLPSmActiveCommonPrio						: BYTE;																								//Loop to check the smalest active common priority
	bySmGrActiveCommonPrio						: BYTE;																								//Smalest or greatest active common priority of the devices
	bySearchBigestPrio							: BYTE;																								//Search the biggest Prio for each device in the Steps in what we choose the prio
	uiState										: UINT;																								//Actual State
	uiState_CP									: UINT;																								//Actual State to compare for activating the timout timer
	diNumberOfDevicesFromEachType				: DINT;																								//Count the Number of each Device what has a priority <> 0
	diMemCmpOperationState						: DINT;																								//Variable to compare the operation state			
	diNumberOfActiveBatterys					: DINT;																								//Number of active batterys
	diNumberOfBatteryInverterInEPO				: DINT;																								//Number of battery inverters that work in Emergency Power operation 
	diNrOfEM_IN_CS_CP							: DINT;																								//Number of the electric meter for receive data. (Its for the complete consumption of all charging stations to compare)
	diNumberOfECS								: DINT;																								//Number of total charging stations on what the power must reduced with the max fuse power
	diBiggestNumberOfDeviceConstants			: DINT;																								//Biggest Number of the constants for the several device types. Needs to calcualte the delay for the timout timer
	dwSumSOC									: DWORD;																							//Sum of the SOC from all batterys
	dwSumSOCInEPO								: DWORD;																							//Sum of the SOC from all batterys that make a island mode at the moment
	dwAvarageBatterySOC							: DWORD;																							//Actual avarage Battery SOC from each Battery
	dwAvarageBatterySOCInEPO					: DWORD;																							//Actual avarage Battery SOC from each Battery that make a island mode at the moment
	udiCounterOnlineChange_CP					: UDINT;																							//Counter for online change to comapre it	
	udiCycleTime								: UDINT;																							//Cycle time in wich the function is running. Needs to calculate the delay for the timout timer
	rValuePercentToControllableDevices			: REAL;																								//Percent value to set the target power to controllable devices
	rValuePercentToStepSwitchedDevices			: REAL;																								//Percent value to set the target power to on/off or step switched devices
	rControllerQPIDSC							: REAL;																								//Controller output from pid self consumption
	rControllerQPIDEPO							: REAL;																								//Controller output from pid emergency power operation
	rSizeMainFuseCS_CP							: REAL;																								//Size of the main fuse form the charging stations to compare with the original varialbe
	lrTargetPowerCorrectionECS					: LREAL;																							//New Target power for chargign station after correction with max fuse power
	lrPowerDiffFuseECS							: LREAL;																							//Power difference between max fuse power charging station and actual power for all charging stations 
	lrPowerForCalculateECS						: LREAL;																							//Power to calcualte the % for each charging station
	lrGridPower									: LREAL;																							//Grid power in kW
	lrGridPower_CP								: LREAL;																							//Grid power in kW to compare for correction when the backend is controlling the battery
	lrSizeBatteryPowerInEPO						: LREAL;																							//Power in kW of all Battery inverters that are made a island mode at the moment
	lrSizeGridConnection						: LREAL;																							//Size of the complete grid connection
	lrActualSurplusOrConsumption				: LREAL;																							//Actual surplus or consumption in kW
	lrActualSurplusOrConsumptionOld				: LREAL;																							//Old value from last step with surplus or consumption in kW
	lrMaxPowerDevicesWithActualPrio				: LREAL;																							//Actual complete max power from all devices with the same priority
	lrErrorPIDCorrectionBattSC					: LREAL;																							//Limit the Error on the pid controller for discahrge the battery on the self consumption mode
	lrErrorPIDCorrectionBattEPO					: LREAL;																							//Limit the Error on the pid controller for discahrge the battery on the emergency power operation mode
	lrErrorPIDCorrectionBattPLCLM_Dischrg		: LREAL;																							//Limit the Error on the pid controller for discahrge the battery on the load management mode and peak shaving mode
	lrErrorPIDCorrectionBattPLCLM_Chrg			: LREAL;																							//Limit the Error on the pid controller for charge the battery on the load management mode and peak shaving mode
	liCounterCkeckDeviceAndPrio					: LINT;																								//Counter to ckeck the device and Prio in the Steps for HP and EHE. Here we didn't can use a loop regarding performance problems on small PLC
	liNrOfNotDoneDevices						: LINT;																								//Shows the Numer of Devices what are not controlled with the minimum or the maximum power when we have a actual Prio from 1 or 255. That we can set the min reached or max reached Flag
	liLPCheckDeviceAndPrio						: LINT;																								//Loop to ckeck the Number of Devices and the Prio
	liLPGridData								: LINT;																								//Loop to check some grid data
	liLPActualSurplusOrConsumption				: LINT;																								//Loop to check actual surplus or consumption
	liLPBatterysSetupData						: LINT;																								//Loop to copy the setup data from the battery inverters
	liLPBatteryData								: LINT;																								//Loop to check some data from batterys
	liLPSumSOCInEPO								: LINT;																								//Loop to calculate the sum of the SOC from all batterys that buils a island mode at the moment
	liLPInEPO									: LINT;																								//Loop to check if 1 or more battery inverters build a island grid
	liLPCheckMaxPower							: LINT;																								//Loop to ckeck the max power from each device
	liLPSetPercentPower							: LINT;																								//Loop to set the calculatet percetn power to the device
	liLPCorrectionPowerCS						: LINT;																								//Loop to make a correction on the target power from the charging stations in dependence of the max fuse power 
	liLPDataBatteryInverter						: LINT;																								//Loop to check or set data from battery inverters
	RS_BatteryChargingControl: RS;
	mtest1: BOOL;
	mtest2: BOOL;
	mTest3: BOOL;
	x: REAL:=0.1;
	y: REAL:=0.01;
	m_fbPIDDischrgCmdFromBackend_Enable: BOOL;
	m_fbPIDBatteryEPO_Enable: BOOL;
	m_fbPIDBatteryPLCLM_Chrg_Enable: BOOL;
	m_fbPIDBatteryPLCLM_Dischrg_Enable:BOOL;
	m_fbPIDBatterySC_Enable: BOOL;

	r_P_Discharge: REAL:=0.04;
	udint_I_Discharge: UDINT := 500;
	udint_D_Discharge: UDINT;
END_VAR

// Zeile 116			bStopAll := FALSE;				gehört gelöst


//Creator : Kai Ebensperger + add on Stefan  V2.0.0.1
//Company : Lynus AG
//Date : 29.05.2021
//Version : 2.0.0.1

//With this FB the EMS control can be realized on the PLC. 
//This divides the excess energy among the devices according to priority
//Devices with priority 0 received as target power 0
//If we have less or no surplus, then the target power will be reduced or remains on the same value
//The EMS function can handle batterie devices, controllable devices, On/Off devices and step switched devices. 
//If we have no surplus, and all devices has a target power from 0, then the battery try to balancing the consumption.
//This depends what operation mode is active
//If the mode load managemant is active, for the charging station the max power from the fuse is neccessary, because the ems dont can use all the power from the max. grid power for the charging stations.  
//When a Batteryinverter or Batterysystem is in Island mode, then ems send to this system automatic -100%. The rest must be regulate the function from the batteryinverter. 
//All other battery inverters or battery systems that do not do islanding are treated by the EMS as normal devices with their priorities.
//This EMS can handle 5 device types (Battery, Heating Pump, Electric heating element, Electric charging station and other big consumers)
//This Function receive also Data from a Backend System. In this Backend System runs different ML-Models.
//So its possible that the Backend System controlls the Heating Pumps when its neccessary and also the discharging from the Batterys.
//This make sense when we have bad wheater, less PV-power in the next 24h to switch on the Heating Pumps or cover the consumption.......
//This EMS Function work only with our Backend Communication Library. After 11 Days no communication to our Backend system or no received new HB the Function dissable automatically and set a Message for this at the output
//When we receiven no HB, no Backend Service Ready Flag or an Error from the Backend Service then the Controlling over the Backend is dissabled and the EMS Function run in his "normal" Mode.

//NOTE for diNr.....Designation => 
//_IN = Here Data come in from other Functions or go out to other functions about the GVL
//_OUT = Here Data go out to other functions about the GVL

// V2.0.0.1
// added option b_ZeroPowerRegulation (Line 1728/1732/1738) 
// added option for disable charging the battery (e.g. for only charging in the night) line 1811 (b_EnableBatteryChargingControl) and 2179 ff(b_EnableBatteryChargingControl,b_StartReleaseBatteryCharging,b_StopReleaseBatteryCharging)
(*------------------------------------------------------------Limits----------------------------------------------------------------------------------*)

stSetupEMS.rSizeMainFuseCS := LIMIT(0,stSetupEMS.rSizeMainFuseCS,500);
	stSetupEMS.uiUpdateTime := LIMIT(1,stSetupEMS.uiUpdateTime,600);
		stSetupEMS.byResChrgfromGridToBatt := LIMIT(0,stSetupEMS.byResChrgfromGridToBatt,100);
			diNrOfEM_IN_ECS := LIMIT(0,diNrOfEM_IN_ECS,Constants_Energy.diMaxNumberOfElectricMeters);
				rHeartbeat := LIMIT(0,rHeartbeat,1);
					rErrorWarning := LIMIT(0,rErrorWarning,2);
						rEnergyOptReady := LIMIT(0,rEnergyOptReady,1);
							rNewBattPower := LIMIT(0,rNewBattPower,100000);				
								rMaxBattChargingPower := LIMIT(0,rMaxBattChargingPower,100);
									rPeakDetectionforCalculation := LIMIT(3,rPeakDetectionforCalculation,100); 

stSetupEMS.rSizeMainFuseCS := DINT_TO_REAL(REAL_TO_DINT(stSetupEMS.rSizeMainFuseCS * 10)) / 10;
		
IF stSetupEMS.byMaxDepthOfDischrgEPO > stSetupEMS.byReserveSOCEPO THEN stSetupEMS.byReserveSOCEPO := stSetupEMS.byMaxDepthOfDischrgEPO + 1; END_IF
	IF stSetupEMS.byMaxDepthOfDischrgEPO > stSetupEMS.byPrioMinChrgBattSOCInEPO THEN stSetupEMS.byPrioMinChrgBattSOCInEPO := stSetupEMS.byMaxDepthOfDischrgEPO + 1; END_IF
		IF stSetupEMS.byReserveSOCEPO > stSetupEMS.byPrioMinChrgBattSOCInEPO THEN stSetupEMS.byPrioMinChrgBattSOCInEPO := stSetupEMS.byReserveSOCEPO + 1; END_IF
		
stSetupEMS.byMaxDepthOfDischrgEPO := LIMIT(0,stSetupEMS.byMaxDepthOfDischrgEPO,100);
	stSetupEMS.byReserveSOCEPO := LIMIT(0,stSetupEMS.byReserveSOCEPO,100);
		stSetupEMS.byPrioMinChrgBattSOCInEPO := LIMIT(20,stSetupEMS.byPrioMinChrgBattSOCInEPO,75);

(*-------------------------------------------------------------Calcualte the number of EMS---------------------------------------------------------------*)

//Online change
timDelayStart(IN:= udiCounterOnlineChange_CP <> TwinCAT_SystemInfoVarList._AppInfo.OnlineChangeCnt, PT:= T#15S, Q=> , ET=> );

fbNumberDevice(
	diActualNumberOfDevices:= Lynus_Standards.GVL_Energy.stNumberOfDevices.diNumberOfEMS, 
	diMaxNumberOfDevices:= Constants_Energy.diMaxNumberOfEMS, 
	udiCounterOnlineChange:= TwinCAT_SystemInfoVarList._AppInfo.OnlineChangeCnt, 
	bNumberIsCalculatet=> , 
	bFPNumberIsCalculatet=> , 
	bOnlineChange=> , 
	diNumberForThisDevice=> diNrOfEMS_OUT, 
	diNumberOfTotalDevices=> );

//Write new Numer on GVL
IF fbNumberDevice.bFPNumberIsCalculatet THEN
	Lynus_Standards.GVL_Energy.stNumberOfDevices.diNumberOfEMS := fbNumberDevice.diNumberOfTotalDevices;	
END_IF 

//Delete old Number on GVL
IF fbNumberDevice.bOnlineChange THEN 
	Lynus_Standards.GVL_Energy.stNumberOfDevices.diNumberOfEMS := diNrOfEMS_OUT;	
		udiCounterOnlineChange_CP := TwinCAT_SystemInfoVarList._AppInfo.OnlineChangeCnt; 
END_IF

(*-------------------------------------------------------------Service from Backend is ready and check the connection to backen for dissabel/enable EMS Function---------------------------------------------------------------*)

//Try to reset the variable for connection on the GVL. When all is normal then the Lynus Mqtt connection function set this variable to true in the next cycle
//When we have no connection to the backend or no HB from the Service then after Lynus_Standards.Constants_General.tTimeDissableLynusFunctions days the EMS is dissabled with all of his functionalities
timResetConnectionOnGVL(IN:= NOT timResetConnectionOnGVL.Q, PT:= T#1H, Q=> , ET=> );
	IF timResetConnectionOnGVL.Q THEN Lynus_Standards.GVL_Communicator.bStateConnectionToEnableFunctions := FALSE; END_IF
		IF NOT Lynus_Standards.GVL_Communicator.bStateConnectionToEnableFunctions OR rHeartbeat_CP = rHeartbeat THEN timDissableFunctions.IN := TRUE; ELSE timDissableFunctions.IN := FALSE; END_IF  
			timDissableFunctions(IN:= , PT:= Lynus_Standards.Constants_General.tTimeDissableLynusFunctions, Q=> , ET=> );
	
//Heartbeat, Service Ready and ErrorWarning from Service
timHB(IN:= , PT:= T#130S, Q=> , ET=> );	
	IF rHeartbeat <> rHeartbeat_CP THEN 
		timHB.IN := FALSE; rHeartbeat_CP := rHeartbeat; 
	ELSE 
		timHB.IN := TRUE; 
	END_IF

//Error/Warning Timer and Service Ready Timer
timErrorWarning(IN:= rErrorWarning = 0, PT:= T#10S, Q=> , ET=> );
	timEnergyOptReady(IN:= rEnergyOptReady <> 0, PT:= T#10S, Q=> , ET=> );
		timControlingState(IN:= bControllingState, PT:= T#10S, Q=> , ET=> );
	
IF timErrorWarning.Q AND timEnergyOptReady.Q AND NOT bControllingState AND NOT timHB.Q AND NOT timDissableFunctions.Q THEN bDischrgCmdFromBackendOK := TRUE; END_IF
	IF rErrorWarning <> 0 OR rEnergyOptReady = 0 OR timControlingState.Q OR timHB.Q OR timDissableFunctions.Q OR NOT bEnable OR eOperationMode = E_OperatingMode_EMS.eAllOff THEN bDischrgCmdFromBackendOK := FALSE; END_IF
	
(*-------------------------------------------------------------Check the number of the device types what are neccessary for EMS---------------------------------------------------------------*)	
	
